// TwinCAT 3 PLC project PLC
// ProgramVersion: 3.1.4023.0
// libraries:
//   Tc2_Standard, * (Beckhoff Automation GmbH)
//   Tc2_System, * (Beckhoff Automation GmbH)
//   Tc3_Module, * (Beckhoff Automation GmbH)
// project tree:
//   / PlcTask.TcTTO
//   POUs/ MAIN.TcPOU
//   DUTs/IO/PdoEntries/ Status_B8381171.TcDUT, Status_182674C6.TcDUT, Status_7097155E.TcDUT, Control_DAEE1D52.TcDUT, Control_F189B737.TcDUT, Control_7786EF9F.TcDUT, Status_70E023F8.TcDUT, Control_A8DDCD82.TcDUT, Status_F2CE6D91.TcDUT, Status_B0753356.TcDUT, Status_68C33E99.TcDUT, Status_ACC8459F.TcDUT, Status_C03E2495.TcDUT, Status_D8D782C3.TcDUT, Control_6EF2C5D0.TcDUT, Status_3E6F3FF3.TcDUT, Status_3D84275F.TcDUT, Ctrl_1EFB4D3B.TcDUT, Status_B6795845.TcDUT, Control_C948E0F2.TcDUT, Status_8CBE219F.TcDUT, Status_1E008DB9.TcDUT, Control_5FD4673D.TcDUT, Status_3035BE2E.TcDUT, Status_2569232E.TcDUT, Control_FF5AB9B2.TcDUT, FSOE_1F44E1B4.TcDUT, FSOE_9A7ED3DD.TcDUT, FSOE_9F04885D.TcDUT, FSOE_87848461.TcDUT, FSOE_BBC930F7.TcDUT, FSOE_D1C9D1EA.TcDUT, FSOE_D94E700C.TcDUT, FSOE_1DB604F4.TcDUT, FSOE_046F804E.TcDUT, FSOE_2DC96D31.TcDUT
//   DUTs/IO/PDOs/ InfoData_6F19DB2B.TcDUT, WcState_0B2B16F9.TcDUT, InfoData_32EB74EA.TcDUT, Channel_830843C1.TcDUT, WcState_9091E0EB.TcDUT, Channel_42CA91F7.TcDUT, PWM_Outputs_Channel_4C6289CD.TcDUT, PTO_Status_E0EB10E8.TcDUT, ENC_Status_compact_3C6E2C44.TcDUT, PLS_Status_Channel_70E7A1E2.TcDUT, PTO_Control_9287F8E4.TcDUT, PTO_Target_compact_5C359F7D.TcDUT, ENC_Control_compact_2E82BC43.TcDUT, PLS_Control_compact_Channel_CD6E44DE.TcDUT, PTO_Status_Channel_E0EB10E8.TcDUT, ENC_Status_Channel_A9252C48.TcDUT, PTO_Control_Channel_9287F8E4.TcDUT, PTO_Target_Channel_1F6D5BC6.TcDUT, ENC_Control_Channel_686BB9DC.TcDUT, AI_Standard_Channel_4A394481.TcDUT, AI_Standard_Channel_A8DF64E3.TcDUT, RTD_Inputs_Channel_9575FEA1.TcDUT, TC_Channel_9575FEA1.TcDUT, AO_Output_Channel_BA7EBB7C.TcDUT, SSI_Inputs_Channel_0E3D8E33.TcDUT, SSI_Inputs_Channel_EDA16284.TcDUT, ENC_Status_compact_7D3464F3.TcDUT, ENC_Control_compact_21E2D14D.TcDUT, ENC_Inputs_B3536485.TcDUT, ENC_Inputs_24B63C53.TcDUT, ENC_Outputs_21E2D14D.TcDUT, COM_Inputs_Channel_3801C95E.TcDUT, COM_Outputs_Channel_EADA2E0D.TcDUT, DeviceState_Inputs_Device_A1210598.TcDUT, DeviceState_Inputs_4751FF76.TcDUT, InfoData_90184F0C.TcDUT, Module_1_DeviceState_Inputs_Device_5322301C.TcDUT, Module_2_DeviceState_Inputs_BD6C7035.TcDUT, STM_Status_36ED096F.TcDUT, STM_Control_5A8B5016.TcDUT, STM_Velocity_A47A3F41.TcDUT, InfoData_6538CF5F.TcDUT, ENC_Status_compact_4D066E1A.TcDUT, STM_Status_DE0D6B37.TcDUT, STM_Control_BA4CE352.TcDUT, ENC_Status_compact_Channel_DC559AB0.TcDUT, DCM_Status_Channel_36ED096F.TcDUT, ENC_Control_compact_Channel_2E82BC43.TcDUT, DCM_Control_Channel_5A8B5016.TcDUT, DCM_Velocity_Channel_A47A3F41.TcDUT, InfoData_939F71B6.TcDUT, FB_Position_3FA094ED.TcDUT, DRV_Statusword_9B36FDFC.TcDUT, DRV_Controlword_F3F14721.TcDUT, DRV_Target_velocity_08A9583B.TcDUT, InfoData_96C94FAE.TcDUT, InfoData_6185D47C.TcDUT, DS402_Statusword_9B36FDFC.TcDUT, DS402_Position_actual_value_07DC4C74.TcDUT, DS402_Controlword_F3F14721.TcDUT, DS402_Target_velocity_08A9583B.TcDUT, InfoData_8300A75E.TcDUT, DCM_Status_Channel_45521CDC.TcDUT, DCM_Outputs_Channel_F77F51CE.TcDUT, DRV_Following_error_actual_value_5AA320BF.TcDUT, DRV_Target_position_05240F14.TcDUT, Status_Uo_B8D9F2FA.TcDUT, BCT_Inputs_8E55234D.TcDUT, BCT_Inputs_4B987895.TcDUT, BCT_Inputs_8B1D510C.TcDUT, BCT_Inputs_7ACE8FA6.TcDUT, FSoE_Inputs_8952FEF0.TcDUT, FSoE_Outputs_7E672439.TcDUT, FIELDVOLTAGE_Field_Voltage_Status_9DC7C349.TcDUT, FSLOGIC_Inputs_EEE9388E.TcDUT, EMPTY_STRUCTURE.TcDUT, Module_1_FSOE_5515F18A.TcDUT, Module_2_DEVICEIO_5FA6B4E7.TcDUT, Module_3_FSLOGIC_DEAB4522.TcDUT, FSoE_Inputs_C661B78A.TcDUT, FSoE_Outputs_E138FCB5.TcDUT, Module_1_FSOE_18ED951F.TcDUT, FSoE_Inputs_8A5FBAF8.TcDUT, FSoE_Outputs_1F40D103.TcDUT, Outputs_7EDA7A42.TcDUT, WcState_B516A264.TcDUT, Module_1_FSOE_9FCACE14.TcDUT, Module_2_FSOUT_5A5AEBA4.TcDUT, Module_3_DEVICEIO_5FA6B4E7.TcDUT, Module_4_FSLOGIC_DEAB4522.TcDUT, FSoE_Inputs_15C2E7B1.TcDUT, FSoE_Outputs_C9D9BEFD.TcDUT, Module_1_FSOE_212A0B66.TcDUT, FSoE_Inputs_939ABF3D.TcDUT, FSoE_Outputs_2DD09AA7.TcDUT, Outputs_FB9F3520.TcDUT, Module_1_FSOE_7F12D292.TcDUT, Module_2_FSOUT_9813A38E.TcDUT, InfoData_E68C61CD.TcDUT, InfoData_2A97D6CF.TcDUT, Inputs_25A0042B.TcDUT, Outputs_2397A10E.TcDUT
//   DUTs/IO/Boxes/ EK1100_1FC0878B.TcDUT, EK1122_1FC0878B.TcDUT, EJ1100_1FC0878B.TcDUT, EJ1101_D4DF6A22.TcDUT, EJ1008_78E8D3DD.TcDUT, EJ1128_78E8D3DD.TcDUT, EJ1809_32157CFD.TcDUT, EJ1819_32157CFD.TcDUT, EJ1859_7699BCF6.TcDUT, EJ1889_32157CFD.TcDUT, EJ1122_1FC0878B.TcDUT, EJ2008_E2806B95.TcDUT, EJ2128_E2806B95.TcDUT, EJ2502_FE2154F7.TcDUT, EJ2521_E6A3E301.TcDUT, EJ2522_EF4C90EB.TcDUT, EJ2809_2B6483BD.TcDUT, EJ2889_2B6483BD.TcDUT, EJ3004_C4269E32.TcDUT, EJ3048_335F857B.TcDUT, EJ3058_335F857B.TcDUT, EJ3068_335F857B.TcDUT, EJ3104_DCC78662.TcDUT, EJ3108_335F857B.TcDUT, EJ3108_35AE5324.TcDUT, EJ3202_27F12237.TcDUT, EJ3214_8BBE23EA.TcDUT, EJ3255_1972F7C0.TcDUT, EJ3318_BD104D88.TcDUT, EJ4002_11E38659.TcDUT, EJ4002_5AE37D91.TcDUT, EJ4004_AB92710E.TcDUT, EJ4008_4E77D882.TcDUT, EJ4018_4E77D882.TcDUT, EJ4024_AB92710E.TcDUT, EJ4132_11E38659.TcDUT, EJ4134_15C7AA14.TcDUT, EJ5002_6DCBC4C0.TcDUT, EJ5002_31A396E2.TcDUT, EJ5101_7476E948.TcDUT, EJ5151_905C5FD8.TcDUT, EJ6002_D5B468BD.TcDUT, EJ6224_98EF2419.TcDUT, EJ7031_022B4804.TcDUT, EJ7037_3E4BEAEF.TcDUT, EJ7041_022B4804.TcDUT, EJ7047_3E4BEAEF.TcDUT, EJ7342_2AE9C6B3.TcDUT, EJ7211_CE650BCF.TcDUT, EJ7211_FC4732E8.TcDUT, EJ7211_7BF21317.TcDUT, EJ7211_B7F6AF53.TcDUT, EJ7334_80FE8C13.TcDUT, EJ7411_236AD61B.TcDUT, EJ9001_1FC0878B.TcDUT, EJ9505_19A4723D.TcDUT, EJ9576_6D7359CA.TcDUT, EJ9576_85AB5804.TcDUT, EJ9576_1017F4A5.TcDUT, EJ9576_C42142C6.TcDUT, EJ9400_B5091FDC.TcDUT, EJ9404_A60D6900.TcDUT, EJ1914_0821024F.TcDUT, EJ1918_57845E79.TcDUT, EJ1957_9A95FC59.TcDUT, EJ2914_475777A0.TcDUT, EJ2918_B661C90A.TcDUT, EJ6910_CD4DE200.TcDUT
//   DUTs/IO/Devices/ SyncUnitTask_2D604ED5.TcDUT, SyncUnitTasks_6FEB8257.TcDUT, SyncUnits_99E584AF.TcDUT
//   DUTs/IO/Topology/ Beckhoff_EJ1xxxEK1122_25307691.TcDUT, Beckhoff_EJ1xxx_8ABA4DFB.TcDUT, Beckhoff_EJ2xxxEK1122_536A6829.TcDUT, Beckhoff_EJ2xxx_F745D3BC.TcDUT, Beckhoff_EJ3xxxEK1122_1A5DA9A5.TcDUT, Beckhoff_EJ3xxx_05F253C1.TcDUT, Beckhoff_EJ4xxxEK1122_E11BF0B6.TcDUT, Beckhoff_EJ4xxx_77B5C5A6.TcDUT, Beckhoff_EJ5xxxEK1122_A82C313A.TcDUT, Beckhoff_EJ5xxx_E1A62FB7.TcDUT, Beckhoff_EJ6xxxEK1122_737473AE.TcDUT, Beckhoff_EJ6xxx_D380D5DE.TcDUT, Beckhoff_EJ7xxxEK1122_3A43B222.TcDUT, Beckhoff_EJ7xxx_D0F87F47.TcDUT, Beckhoff_EJ9xxxEK1122_C80E1DB3.TcDUT, Beckhoff_EJ9xxx_428E1E12.TcDUT, Beckhoff_EJx9xxEK1122_EEA9E9F5.TcDUT, Beckhoff_EJx9xx_66D9432D.TcDUT, EtherCAT_Master_EJxxxx_F8B494BA.TcDUT
//   DUTs/IO/Base/ EtcSlaveBase_82538BE2.TcDUT, EtcSlaveBase_82538BE2.TcDUT, EtcSlaveBase_82538BE2.TcDUT, EtcSlaveTerminalBase_947E5A46.TcDUT, EtcSlaveBoxBase_77A0E4A7.TcDUT, EtcSlaveEndTerminalBase_866C7F0C.TcDUT, InputBase_8311D824.TcDUT, OutputBase_10CEE7DE.TcDUT, EtcMasterBase_62654B43.TcDUT
//   GVLs/ GVL_iXlinker.TcGVL
// real-time tasks:
//   TASK PlcTask: cycle T#10ms, priority 20, ADS port 350
// I/O:
//   DEVICE EtherCAT_Master_EJxxxx, AmsNetId 172.20.30.238.7.1
//     Beckhoff EJ1xxx [EK1100 EtherCAT Coupler (2A E-Bus)]
//       Beckhoff EJ1xxxEK1122 [EK1122 2 port EtherCAT junction]
//         Beckhoff EJ1xxxsub EK1100 [EK1100 EtherCAT Coupler (2A E-Bus)]
//         A_0001(EJ1100-0000-0018) [EJ1100 EtherCAT Coupler (2.2A E-Bus)]
//         A_0002(EJ1101-0022-0016) [EJ1101-0022 EtherCAT Coupler (ID switch)]
//       A_0004(EJ1008-0000-0017) [EJ1008 8Ch. Dig. Input 24V, 3ms]
//       A_0005(EJ1128-0000-0016) [EJ1128 8Ch. Dig. Input 5V / 3.3V DC, 0.05µs]
//       A_0006(EJ1809-0000-0017) [EJ1809 16Ch. Dig. Input 24V, 3ms]
//       A_0007(EJ1819-0000-0017) [EJ1819 16Ch. Dig. Input 24V, 10µs]
//       A_0008(EJ1859-0000-0017) [EJ1859 8Ch. Dig. Input 24V, 3ms, 8Ch. Dig. Output 24V, 0.5A]
//       A_0009(EJ1889-0000-0017) [EJ1889 16Ch. Dig. Input 24V, 3ms, negative]
//       A_0003(EJ1122-0000-0016) [EJ1122 2 port EtherCAT junction]
//     Beckhoff EJ2xxx [EK1100 EtherCAT Coupler (2A E-Bus)]
//       Beckhoff EJ2xxxEK1122 [EK1122 2 port EtherCAT junction]
//         Beckhoff EJ2xxxsub EK1100 [EK1100 EtherCAT Coupler (2A E-Bus)]
//       A_0001(EJ2008-0000-0017) [EJ2008 8Ch. Dig. Output 24V, 0.5A]
//       A_0002(EJ2008-0000-0018) [EJ2008 8Ch. Dig. Output 24V, 0.5A]
//       A_0003(EJ2128-0000-0016) [EJ2128 8Ch. Dig. Output 5V/3.3V, 20mA]
//       A_0004(EJ2502-0000-0023) [EJ2502 2Ch. PWM output, 24V]
//       A_0005(EJ2502-0000-0024) [EJ2502 2Ch. PWM output, 24V]
//       A_0006(EJ2521-0224-0016) [EJ2521-0224 1Ch. Pulse Train 24V DC Output Capture/Compare]
//       A_0007(EJ2522-0000-0022) [EJ2522 2Ch. Pulse Train Output]
//       A_0008(EJ2809-0000-0017) [EJ2809 16Ch. Dig. Output 24V, 0.5A]
//       A_0009(EJ2889-0000-0016) [EJ2889 16Ch. Dig. Output 24V, 0.5A, negative]
//       A_0010(EJ2889-0000-0017) [EJ2889 16Ch. Dig. Output 24V, 0.5A, negative]
//     Beckhoff EJ3xxx [EK1100 EtherCAT Coupler (2A E-Bus)]
//       Beckhoff EJ3xxxEK1122 [EK1122 2 port EtherCAT junction]
//         Beckhoff EJ3xxxsub EK1100 [EK1100 EtherCAT Coupler (2A E-Bus)]
//       A_0001(EJ3004-0000-0019) [EJ3004 4Ch. Ana. Input +/-10V]
//       A_0002(EJ3004-0000-0020) [EJ3004 4Ch. Ana. Input +/-10V]
//       A_0003(EJ3004-0000-0021) [EJ3004 4Ch. Ana. Input +/-10V]
//       A_0004(EJ3048-0000-0020) [EJ3048 8Ch. Ana. Input 0-20mA]
//       A_0005(EJ3058-0000-0020) [EJ3058 8Ch. Ana. Input 4-20mA]
//       A_0006(EJ3068-0000-0020) [EJ3068 8Ch. Ana. Input 0-10V]
//       A_0007(EJ3068-0000-0021) [EJ3068 8Ch. Ana. Input 0-10V]
//       A_0008(EJ3104-0000-0019) [EJ3104 4Ch. Ana. Input +/-10V DIFF]
//       A_0009(EJ3104-0000-0020) [EJ3104 4Ch. Ana. Input +/-10V DIFF]
//       A_0010(EJ3104-0000-0021) [EJ3104 4Ch. Ana. Input +/-10V DIFF]
//       A_0011(EJ3108-0000-0017) [EJ3108 8Ch. Ana. Input +/-10V]
//       A_0012(EJ3108-0000-0018) [EJ3108 8Ch. Ana. Input +/-10V]
//       A_0013(EJ3108-0000-0019) [EJ3108 8Ch. Ana. Input +/-10V]
//       A_0014(EJ3202-0000-0019) [EJ3202 2Ch. Ana. Input PT100 (RTD)]
//       A_0015(EJ3202-0000-0020) [EJ3202 2Ch. Ana. Input PT100 (RTD)]
//       A_0016(EJ3202-0000-0021) [EJ3202 2Ch. Ana. Input PT100 (RTD)]
//       A_0017(EJ3214-0000-0016) [EJ3214 4Ch. Ana. Input PT100 (RTD)]
//       A_0018(EJ3255-0000-0023) [EJ3255 5Ch. potentiometer measurement with sensor supply]
//       A_0019(EJ3318-0000-0017) [EJ3318 8Ch. Ana Input Thermocouple (TC)]
//     Beckhoff EJ4xxx [EK1100 EtherCAT Coupler (2A E-Bus)]
//       Beckhoff EJ4xxxEK1122 [EK1122 2 port EtherCAT junction]
//         Beckhoff EJ4xxxsub EK1100 [EK1100 EtherCAT Coupler (2A E-Bus)]
//       A_0001(EJ4002-0000-0017) [EJ4002 2Ch. Ana. Output 0-10V, 12bit]
//       A_0002(EJ4002-0000-0018) [EJ4002 2Ch. Ana. Output 0-10V, 12bit]
//       A_0003(EJ4004-0000-0020) [EJ4004 4Ch. Ana. Output 0-10V, 12bit]
//       A_0004(EJ4008-0000-0020) [EJ4008 8Ch. Ana. Output 0-10V, 12bit]
//       A_0005(EJ4018-0000-0016) [EJ4018 8Ch. Ana. Output 0-20mA, 12bit]
//       A_0006(EJ4024-0000-0020) [EJ4024 4Ch. Ana. Output 4-20mA, 12bit]
//       A_0007(EJ4132-0000-0019) [EJ4132 2Ch. Ana. Output -10/+10V, 16bit]
//       A_0008(EJ4134-0000-0019) [EJ4134 4Ch. Ana. Output -10/+10V, 16bit]
//       A_0009(EJ4134-0000-0020) [EJ4134 4Ch. Ana. Output -10/+10V, 16bit]
//     Beckhoff EJ5xxx [EK1100 EtherCAT Coupler (2A E-Bus)]
//       Beckhoff EJ5xxxEK1122 [EK1122 2 port EtherCAT junction]
//         Beckhoff EJ5xxxsub EK1100 [EK1100 EtherCAT Coupler (2A E-Bus)]
//       A_0001(EJ5002-0000-0016) [EJ5002 2Ch. SSI Encoder]
//       A_0002(EJ5002-0000-0017) [EJ5002 2Ch. SSI Encoder]
//       A_0003(EJ5101-0000-0016) [EJ5101 1Ch. Inc. Encoder 5V]
//       A_0004(EJ5151-0000-0016) [EJ5151 1Ch. Inc. Encoder]
//     Beckhoff EJ6xxx [EK1100 EtherCAT Coupler (2A E-Bus)]
//       Beckhoff EJ6xxxEK1122 [EK1122 2 port EtherCAT junction]
//         Beckhoff EJ6xxxsub EK1100 [EK1100 EtherCAT Coupler (2A E-Bus)]
//       A_0001(EJ6002-0000-0016) [EJ6002 Interface 2Ch. (RS232/RS485/RS422)]
//       A_0002(EJ6224-0000-0016) [EJ6224 (IO Link Master)]
//         modules: Module 1 (DeviceState Inputs Device), Module 2 (DeviceState Inputs), Module 3 (empty), Module 4 (empty), Module 5 (empty), Module 6 (empty)
//       A_0003(EJ6224-0090-0016) [EJ6224-0090 (IO Link Master, TwinSAFE SC)]
//         modules: Module 1 (DeviceState Inputs Device), Module 2 (DeviceState Inputs), Module 3 (empty), Module 4 (empty), Module 5 (empty), Module 6 (empty)
//     Beckhoff EJ7xxx [EK1100 EtherCAT Coupler (2A E-Bus)]
//       Beckhoff EJ7xxxEK1122 [EK1122 2 port EtherCAT junction]
//         Beckhoff EJ7xxxsub EK1100 [EK1100 EtherCAT Coupler (2A E-Bus)]
//       A_0001(EJ7031-0000-0026) [EJ7031 1Ch. Stepper motor output stage (24V, 1.5A)]
//       A_0002(EJ7037-0000-0020) [EJ7037 1Ch. Stepper motor output stage (24V, 1.5A)]
//       A_0003(EJ7041-0052-0016) [EJ7041-0052 1Ch. Stepper motor output stage (50V, 5A)]
//       A_0004(EJ7047-0000-0018) [EJ7047 1Ch. Stepper motor output stage (50V, 5A)]
//       A_0005(EJ7047-0000-0019) [EJ7047 1Ch. Stepper motor output stage (50V, 5A)]
//       A_0006(EJ7047-0000-0020) [EJ7047 1Ch. Stepper motor output stage (50V, 5A)]
//       A_0007(EJ7342-0000-0019) [EJ7342 2Ch. DC motor output stage (50V, 3.5A)]
//       A_0008(EJ7342-0000-0020) [EJ7342 2Ch. DC motor output stage (50V, 3.5A)]
//       A_0009(EJ7211-0010-0026) [EJ7211-0010 1Ch. MDP742 Servo motor output stage with OCT (50V, 4.5A RMS)]
//       A_0010(EJ7211-0010-0027) [EJ7211-0010 1Ch. MDP742 Servo motor output stage with OCT (50V, 4.5A RMS)]
//       A_0011(EJ7211-0010-0028) [EJ7211-0010 1Ch. MDP742 Servo motor output stage with OCT (50V, 4.5A RMS)]
//       A_0012(EJ7211-0010-0029) [EJ7211-0010 1Ch. MDP742 Servo motor output stage with OCT (50V, 4.5A RMS)]
//       A_0013(EJ7211-0010-0030) [EJ7211-0010 1Ch. MDP742 Servo motor output stage with OCT (50V, 4.5A RMS)]
//       A_0014(EJ7211-0010-0031) [EJ7211-0010 1Ch. MDP742 Servo motor output stage with OCT (50V, 4.5A RMS)]
//       A_0015(EJ7211-0010-0032) [EJ7211-0010 1Ch. MDP742 Servo motor output stage with OCT (50V, 4.5A RMS)]
//       A_0016(EJ7211-0011-0026) [EJ7211-0011 1Ch. DS402 Servo motor output stage with OCT (50V, 4.5A RMS)]
//       A_0017(EJ7211-0011-0027) [EJ7211-0011 1Ch. DS402 Servo motor output stage with OCT (50V, 4.5A RMS)]
//       A_0018(EJ7211-0011-0028) [EJ7211-0011 1Ch. DS402 Servo motor output stage with OCT (50V, 4.5A RMS)]
//       A_0019(EJ7211-0011-0029) [EJ7211-0011 1Ch. DS402 Servo motor output stage with OCT (50V, 4.5A RMS)]
//       A_0020(EJ7211-0011-0030) [EJ7211-0011 1Ch. DS402 Servo motor output stage with OCT (50V, 4.5A RMS)]
//       A_0021(EJ7211-0011-0031) [EJ7211-0011 1Ch. DS402 Servo motor output stage with OCT (50V, 4.5A RMS)]
//       A_0022(EJ7211-0011-0032) [EJ7211-0011 1Ch. DS402 Servo motor output stage with OCT (50V, 4.5A RMS)]
//       A_0023(EJ7211-9414-0029) [EJ7211-9414 1Ch. MDP742 Servo motor output stage with OCT (50V, 4.5A RMS) , TwinSAFE SC]
//       A_0024(EJ7211-9414-0030) [EJ7211-9414 1Ch. MDP742 Servo motor output stage with OCT (50V, 4.5A RMS) , TwinSAFE SC]
//       A_0025(EJ7211-9414-0031) [EJ7211-9414 1Ch. MDP742 Servo motor output stage with OCT (50V, 4.5A RMS) , TwinSAFE SC]
//       A_0026(EJ7211-9414-0032) [EJ7211-9414 1Ch. MDP742 Servo motor output stage with OCT (50V, 4.5A RMS) , TwinSAFE SC]
//       A_0027(EJ7211-9415-0029) [EJ7211-9415 1Ch. DS402 Servo motor output stage with OCT (50V, 4.5A RMS), TwinSAFE SC]
//       A_0028(EJ7211-9415-0030) [EJ7211-9415 1Ch. DS402 Servo motor output stage with OCT (50V, 4.5A RMS), TwinSAFE SC]
//       A_0029(EJ7211-9415-0031) [EJ7211-9415 1Ch. DS402 Servo motor output stage with OCT (50V, 4.5A RMS), TwinSAFE SC]
//       A_0030(EJ7211-9415-0032) [EJ7211-9415 1Ch. DS402 Servo motor output stage with OCT (50V, 4.5A RMS), TwinSAFE SC]
//       A_0031(EJ7334-0008-0016) [EJ7334-0008 4 Ch. Bi-/8 Ch. Unidirectional DC motor output stage (24 V, 8 A overall current)]
//       A_0032(EJ7411-0000-0018) [EJ7411 BLDC Terminal with incremental encoder/Hall, 50 V DC, 4.5 A]
//     Beckhoff EJ9xxx [EK1100 EtherCAT Coupler (2A E-Bus)]
//       Beckhoff EJ9xxxEK1122 [EK1122 2 port EtherCAT junction]
//         Beckhoff EJ9xxxsub EK1100 [EK1100 EtherCAT Coupler (2A E-Bus)]
//       A_0001(EJ9001-0000-0016) [EJ9001 placeholder module]
//       A_0002(EJ9505-0000-0016) [EJ9505 Power supply module 5V]
//       A_0003(EJ9576-0000-0018) [EJ9576 Brake chopper terminal]
//       A_0004(EJ9576-0000-0019) [EJ9576 Brake chopper terminal]
//       A_0005(EJ9576-0000-0020) [EJ9576 Brake chopper terminal]
//       A_0006(EJ9576-0000-0022) [EJ9576 Brake chopper terminal]
//       A_0007 (EJ9400-0000) [EJ9400-0000 Power supply module 2,5A]
//       A_0008 (EJ9404-0000) [EJ9404-0000 Power supply module 12A]
//     Beckhoff EJx9xx [EK1100 EtherCAT Coupler (2A E-Bus)]
//       Beckhoff EJx9xxEK1122 [EK1122 2 port EtherCAT junction]
//         Beckhoff EJx9xxsub EK1100 [EK1100 EtherCAT Coupler (2A E-Bus)]
//       A_0001(EJ1914-0000-0017) [EJ1914-0000-0017]
//         modules: Module 1 (FSOE), Module 2 (DEVICEIO), Module 3 (FSLOGIC)
//       A_0002(EJ1914-0000-0018) [EJ1914, 4Ch. Safety Input 24V, TwinSAFE]
//         modules: Module 1 (FSOE), Module 2 (DEVICEIO), Module 3 (FSLOGIC)
//       A_0003(EJ1918-0000-0017) [EJ1918-0000-0017]
//         modules: Module 1 (FSOE), Module 2 (DEVICEIO), Module 3 (FSLOGIC)
//       A_0004(EJ1918-0000-0018) [EJ1918, 8Ch. Safety Input 24V, TwinSAFE]
//         modules: Module 1 (FSOE), Module 2 (DEVICEIO), Module 3 (FSLOGIC)
//       A_0005(EJ1957-0000-0017) [EJ1957-0000-0017]
//         modules: Module 1 (FSOE), Module 2 (FSOUT), Module 3 (DEVICEIO), Module 4 (FSLOGIC)
//       A_0006(EJ1957-0000-0018) [EJ1957, 8Ch. Safety Input 24V, 4Ch. Safety Output 24V, 0.5A, TwinSAFE]
//         modules: Module 1 (FSOE), Module 2 (FSOUT), Module 3 (DEVICEIO), Module 4 (FSLOGIC)
//       A_0007(EJ2914-0000-0017) [EJ2914-0000-0017]
//         modules: Module 1 (FSOE), Module 2 (FSOUT), Module 3 (DEVICEIO), Module 4 (FSLOGIC)
//       A_0008(EJ2914-0000-0018) [EJ2914, 4Ch. Safety Output 24V, 0.5A, TwinSAFE]
//         modules: Module 1 (FSOE), Module 2 (FSOUT), Module 3 (DEVICEIO), Module 4 (FSLOGIC)
//       A_0009(EJ2918-0000-0017) [EJ2918-0000-0017]
//         modules: Module 1 (FSOE), Module 2 (FSOUT), Module 3 (DEVICEIO), Module 4 (FSLOGIC)
//       A_0010(EJ2918-0000-0018) [EJ2918, 8Ch. Safety Output 24V, 0.5A, TwinSAFE]
//         modules: Module 1 (FSOE), Module 2 (FSOUT), Module 3 (DEVICEIO), Module 4 (FSLOGIC)
//       A_0011(EJ6910-0000-0018) [EJ6910, TwinSAFE PLC]
//       A_0012(EJ6910-0000-0020) [EJ6910, TwinSAFE PLC]
// variable links:
//   PLC/PLC Instance <-> EtherCAT Master EJxxxx/Beckhoff EJ1xxx
//     PlcTask Inputs/GVL_iXlinker.EtherCAT_Master_EJxxxx.Beckhoff_EJ1xxx.InfoData.State <-> InfoData/State
//   PLC/PLC Instance <-> EtherCAT Master EJxxxx/Beckhoff EJ1xxx/Beckhoff EJ1xxxEK1122
//     PlcTask Inputs/GVL_iXlinker.EtherCAT_Master_EJxxxx.Beckhoff_EJ1xxx.Beckhoff_EJ1xxxEK1122.InfoData.State <-> InfoData/State
//   PLC/PLC Instance <-> EtherCAT Master EJxxxx/Beckhoff EJ1xxx/Beckhoff EJ1xxxEK1122/Beckhoff EJ1xxxsub EK1100
//     PlcTask Inputs/GVL_iXlinker.EtherCAT_Master_EJxxxx.Beckhoff_EJ1xxx.Beckhoff_EJ1xxxEK1122.Beckhoff_EJ1xxxsub_EK1100.InfoData.State <-> InfoData/State
//   PLC/PLC Instance <-> EtherCAT Master EJxxxx/Beckhoff EJ1xxx/Beckhoff EJ1xxxEK1122/A_0001(EJ1100-0000-0018)
//     PlcTask Inputs/GVL_iXlinker.EtherCAT_Master_EJxxxx.Beckhoff_EJ1xxx.Beckhoff_EJ1xxxEK1122.A_0001_EJ1100_0000_0018.InfoData.State <-> InfoData/State
//   PLC/PLC Instance <-> EtherCAT Master EJxxxx/Beckhoff EJ1xxx/Beckhoff EJ1xxxEK1122/A_0002(EJ1101-0022-0016)
//     PlcTask Inputs/GVL_iXlinker.EtherCAT_Master_EJxxxx.Beckhoff_EJ1xxx.Beckhoff_EJ1xxxEK1122.A_0002_EJ1101_0022_0016.WcState.WcState <-> WcState/WcState
//     PlcTask Inputs/GVL_iXlinker.EtherCAT_Master_EJxxxx.Beckhoff_EJ1xxx.Beckhoff_EJ1xxxEK1122.A_0002_EJ1101_0022_0016.InfoData.AdsAddr <-> InfoData/AdsAddr
//     PlcTask Inputs/GVL_iXlinker.EtherCAT_Master_EJxxxx.Beckhoff_EJ1xxx.Beckhoff_EJ1xxxEK1122.A_0002_EJ1101_0022_0016.InfoData.State <-> InfoData/State
//   PLC/PLC Instance <-> EtherCAT Master EJxxxx/Beckhoff EJ1xxx/A_0004(EJ1008-0000-0017)
//     PlcTask Inputs/GVL_iXlinker.EtherCAT_Master_EJxxxx.Beckhoff_EJ1xxx.A_0004_EJ1008_0000_0017.Channel_1.Input <-> Channel 1/Input
//     PlcTask Inputs/GVL_iXlinker.EtherCAT_Master_EJxxxx.Beckhoff_EJ1xxx.A_0004_EJ1008_0000_0017.Channel_2.Input <-> Channel 2/Input
//     PlcTask Inputs/GVL_iXlinker.EtherCAT_Master_EJxxxx.Beckhoff_EJ1xxx.A_0004_EJ1008_0000_0017.Channel_3.Input <-> Channel 3/Input
//     PlcTask Inputs/GVL_iXlinker.EtherCAT_Master_EJxxxx.Beckhoff_EJ1xxx.A_0004_EJ1008_0000_0017.Channel_4.Input <-> Channel 4/Input
//     PlcTask Inputs/GVL_iXlinker.EtherCAT_Master_EJxxxx.Beckhoff_EJ1xxx.A_0004_EJ1008_0000_0017.Channel_5.Input <-> Channel 5/Input
//     PlcTask Inputs/GVL_iXlinker.EtherCAT_Master_EJxxxx.Beckhoff_EJ1xxx.A_0004_EJ1008_0000_0017.Channel_6.Input <-> Channel 6/Input
//     PlcTask Inputs/GVL_iXlinker.EtherCAT_Master_EJxxxx.Beckhoff_EJ1xxx.A_0004_EJ1008_0000_0017.Channel_7.Input <-> Channel 7/Input
//     PlcTask Inputs/GVL_iXlinker.EtherCAT_Master_EJxxxx.Beckhoff_EJ1xxx.A_0004_EJ1008_0000_0017.Channel_8.Input <-> Channel 8/Input
//     PlcTask Inputs/GVL_iXlinker.EtherCAT_Master_EJxxxx.Beckhoff_EJ1xxx.A_0004_EJ1008_0000_0017.WcState.WcState <-> WcState/WcState
//     PlcTask Inputs/GVL_iXlinker.EtherCAT_Master_EJxxxx.Beckhoff_EJ1xxx.A_0004_EJ1008_0000_0017.WcState.InputToggle <-> WcState/InputToggle
//     PlcTask Inputs/GVL_iXlinker.EtherCAT_Master_EJxxxx.Beckhoff_EJ1xxx.A_0004_EJ1008_0000_0017.InfoData.State <-> InfoData/State
//   PLC/PLC Instance <-> EtherCAT Master EJxxxx/Beckhoff EJ1xxx/A_0005(EJ1128-0000-0016)
//     PlcTask Inputs/GVL_iXlinker.EtherCAT_Master_EJxxxx.Beckhoff_EJ1xxx.A_0005_EJ1128_0000_0016.Channel_1.Input <-> Channel 1/Input
//     PlcTask Inputs/GVL_iXlinker.EtherCAT_Master_EJxxxx.Beckhoff_EJ1xxx.A_0005_EJ1128_0000_0016.Channel_2.Input <-> Channel 2/Input
//     PlcTask Inputs/GVL_iXlinker.EtherCAT_Master_EJxxxx.Beckhoff_EJ1xxx.A_0005_EJ1128_0000_0016.Channel_3.Input <-> Channel 3/Input
//     PlcTask Inputs/GVL_iXlinker.EtherCAT_Master_EJxxxx.Beckhoff_EJ1xxx.A_0005_EJ1128_0000_0016.Channel_4.Input <-> Channel 4/Input
//     PlcTask Inputs/GVL_iXlinker.EtherCAT_Master_EJxxxx.Beckhoff_EJ1xxx.A_0005_EJ1128_0000_0016.Channel_5.Input <-> Channel 5/Input
//     PlcTask Inputs/GVL_iXlinker.EtherCAT_Master_EJxxxx.Beckhoff_EJ1xxx.A_0005_EJ1128_0000_0016.Channel_6.Input <-> Channel 6/Input
//     PlcTask Inputs/GVL_iXlinker.EtherCAT_Master_EJxxxx.Beckhoff_EJ1xxx.A_0005_EJ1128_0000_0016.Channel_7.Input <-> Channel 7/Input
//     PlcTask Inputs/GVL_iXlinker.EtherCAT_Master_EJxxxx.Beckhoff_EJ1xxx.A_0005_EJ1128_0000_0016.Channel_8.Input <-> Channel 8/Input
//     PlcTask Inputs/GVL_iXlinker.EtherCAT_Master_EJxxxx.Beckhoff_EJ1xxx.A_0005_EJ1128_0000_0016.WcState.WcState <-> WcState/WcState
//     PlcTask Inputs/GVL_iXlinker.EtherCAT_Master_EJxxxx.Beckhoff_EJ1xxx.A_0005_EJ1128_0000_0016.WcState.InputToggle <-> WcState/InputToggle
//     PlcTask Inputs/GVL_iXlinker.EtherCAT_Master_EJxxxx.Beckhoff_EJ1xxx.A_0005_EJ1128_0000_0016.InfoData.State <-> InfoData/State
//   PLC/PLC Instance <-> EtherCAT Master EJxxxx/Beckhoff EJ1xxx/A_0006(EJ1809-0000-0017)
//     PlcTask Inputs/GVL_iXlinker.EtherCAT_Master_EJxxxx.Beckhoff_EJ1xxx.A_0006_EJ1809_0000_0017.Channel_1.Input <-> Channel 1/Input
//     PlcTask Inputs/GVL_iXlinker.EtherCAT_Master_EJxxxx.Beckhoff_EJ1xxx.A_0006_EJ1809_0000_0017.Channel_2.Input <-> Channel 2/Input
//     PlcTask Inputs/GVL_iXlinker.EtherCAT_Master_EJxxxx.Beckhoff_EJ1xxx.A_0006_EJ1809_0000_0017.Channel_3.Input <-> Channel 3/Input
//     PlcTask Inputs/GVL_iXlinker.EtherCAT_Master_EJxxxx.Beckhoff_EJ1xxx.A_0006_EJ1809_0000_0017.Channel_4.Input <-> Channel 4/Input
//     PlcTask Inputs/GVL_iXlinker.EtherCAT_Master_EJxxxx.Beckhoff_EJ1xxx.A_0006_EJ1809_0000_0017.Channel_5.Input <-> Channel 5/Input
//     PlcTask Inputs/GVL_iXlinker.EtherCAT_Master_EJxxxx.Beckhoff_EJ1xxx.A_0006_EJ1809_0000_0017.Channel_6.Input <-> Channel 6/Input
//     PlcTask Inputs/GVL_iXlinker.EtherCAT_Master_EJxxxx.Beckhoff_EJ1xxx.A_0006_EJ1809_0000_0017.Channel_7.Input <-> Channel 7/Input
//     PlcTask Inputs/GVL_iXlinker.EtherCAT_Master_EJxxxx.Beckhoff_EJ1xxx.A_0006_EJ1809_0000_0017.Channel_8.Input <-> Channel 8/Input
//     PlcTask Inputs/GVL_iXlinker.EtherCAT_Master_EJxxxx.Beckhoff_EJ1xxx.A_0006_EJ1809_0000_0017.Channel_9.Input <-> Channel 9/Input
//     PlcTask Inputs/GVL_iXlinker.EtherCAT_Master_EJxxxx.Beckhoff_EJ1xxx.A_0006_EJ1809_0000_0017.Channel_10.Input <-> Channel 10/Input
//     PlcTask Inputs/GVL_iXlinker.EtherCAT_Master_EJxxxx.Beckhoff_EJ1xxx.A_0006_EJ1809_0000_0017.Channel_11.Input <-> Channel 11/Input
//     PlcTask Inputs/GVL_iXlinker.EtherCAT_Master_EJxxxx.Beckhoff_EJ1xxx.A_0006_EJ1809_0000_0017.Channel_12.Input <-> Channel 12/Input
//     PlcTask Inputs/GVL_iXlinker.EtherCAT_Master_EJxxxx.Beckhoff_EJ1xxx.A_0006_EJ1809_0000_0017.Channel_13.Input <-> Channel 13/Input
//     PlcTask Inputs/GVL_iXlinker.EtherCAT_Master_EJxxxx.Beckhoff_EJ1xxx.A_0006_EJ1809_0000_0017.Channel_14.Input <-> Channel 14/Input
//     PlcTask Inputs/GVL_iXlinker.EtherCAT_Master_EJxxxx.Beckhoff_EJ1xxx.A_0006_EJ1809_0000_0017.Channel_15.Input <-> Channel 15/Input
//     PlcTask Inputs/GVL_iXlinker.EtherCAT_Master_EJxxxx.Beckhoff_EJ1xxx.A_0006_EJ1809_0000_0017.Channel_16.Input <-> Channel 16/Input
//     PlcTask Inputs/GVL_iXlinker.EtherCAT_Master_EJxxxx.Beckhoff_EJ1xxx.A_0006_EJ1809_0000_0017.WcState.WcState <-> WcState/WcState
//     PlcTask Inputs/GVL_iXlinker.EtherCAT_Master_EJxxxx.Beckhoff_EJ1xxx.A_0006_EJ1809_0000_0017.WcState.InputToggle <-> WcState/InputToggle
//     PlcTask Inputs/GVL_iXlinker.EtherCAT_Master_EJxxxx.Beckhoff_EJ1xxx.A_0006_EJ1809_0000_0017.InfoData.State <-> InfoData/State
//   PLC/PLC Instance <-> EtherCAT Master EJxxxx/Beckhoff EJ1xxx/A_0007(EJ1819-0000-0017)
//     PlcTask Inputs/GVL_iXlinker.EtherCAT_Master_EJxxxx.Beckhoff_EJ1xxx.A_0007_EJ1819_0000_0017.Channel_1.Input <-> Channel 1/Input
//     PlcTask Inputs/GVL_iXlinker.EtherCAT_Master_EJxxxx.Beckhoff_EJ1xxx.A_0007_EJ1819_0000_0017.Channel_2.Input <-> Channel 2/Input
//     PlcTask Inputs/GVL_iXlinker.EtherCAT_Master_EJxxxx.Beckhoff_EJ1xxx.A_0007_EJ1819_0000_0017.Channel_3.Input <-> Channel 3/Input
//     PlcTask Inputs/GVL_iXlinker.EtherCAT_Master_EJxxxx.Beckhoff_EJ1xxx.A_0007_EJ1819_0000_0017.Channel_4.Input <-> Channel 4/Input
//     PlcTask Inputs/GVL_iXlinker.EtherCAT_Master_EJxxxx.Beckhoff_EJ1xxx.A_0007_EJ1819_0000_0017.Channel_5.Input <-> Channel 5/Input
//     PlcTask Inputs/GVL_iXlinker.EtherCAT_Master_EJxxxx.Beckhoff_EJ1xxx.A_0007_EJ1819_0000_0017.Channel_6.Input <-> Channel 6/Input
//     PlcTask Inputs/GVL_iXlinker.EtherCAT_Master_EJxxxx.Beckhoff_EJ1xxx.A_0007_EJ1819_0000_0017.Channel_7.Input <-> Channel 7/Input
//     PlcTask Inputs/GVL_iXlinker.EtherCAT_Master_EJxxxx.Beckhoff_EJ1xxx.A_0007_EJ1819_0000_0017.Channel_8.Input <-> Channel 8/Input
//     PlcTask Inputs/GVL_iXlinker.EtherCAT_Master_EJxxxx.Beckhoff_EJ1xxx.A_0007_EJ1819_0000_0017.Channel_9.Input <-> Channel 9/Input
//     PlcTask Inputs/GVL_iXlinker.EtherCAT_Master_EJxxxx.Beckhoff_EJ1xxx.A_0007_EJ1819_0000_0017.Channel_10.Input <-> Channel 10/Input
//     PlcTask Inputs/GVL_iXlinker.EtherCAT_Master_EJxxxx.Beckhoff_EJ1xxx.A_0007_EJ1819_0000_0017.Channel_11.Input <-> Channel 11/Input
//     PlcTask Inputs/GVL_iXlinker.EtherCAT_Master_EJxxxx.Beckhoff_EJ1xxx.A_0007_EJ1819_0000_0017.Channel_12.Input <-> Channel 12/Input
//     PlcTask Inputs/GVL_iXlinker.EtherCAT_Master_EJxxxx.Beckhoff_EJ1xxx.A_0007_EJ1819_0000_0017.Channel_13.Input <-> Channel 13/Input
//     PlcTask Inputs/GVL_iXlinker.EtherCAT_Master_EJxxxx.Beckhoff_EJ1xxx.A_0007_EJ1819_0000_0017.Channel_14.Input <-> Channel 14/Input
//     PlcTask Inputs/GVL_iXlinker.EtherCAT_Master_EJxxxx.Beckhoff_EJ1xxx.A_0007_EJ1819_0000_0017.Channel_15.Input <-> Channel 15/Input
//     PlcTask Inputs/GVL_iXlinker.EtherCAT_Master_EJxxxx.Beckhoff_EJ1xxx.A_0007_EJ1819_0000_0017.Channel_16.Input <-> Channel 16/Input
//     PlcTask Inputs/GVL_iXlinker.EtherCAT_Master_EJxxxx.Beckhoff_EJ1xxx.A_0007_EJ1819_0000_0017.WcState.WcState <-> WcState/WcState
//     PlcTask Inputs/GVL_iXlinker.EtherCAT_Master_EJxxxx.Beckhoff_EJ1xxx.A_0007_EJ1819_0000_0017.WcState.InputToggle <-> WcState/InputToggle
//     PlcTask Inputs/GVL_iXlinker.EtherCAT_Master_EJxxxx.Beckhoff_EJ1xxx.A_0007_EJ1819_0000_0017.InfoData.State <-> InfoData/State
//   PLC/PLC Instance <-> EtherCAT Master EJxxxx/Beckhoff EJ1xxx/A_0008(EJ1859-0000-0017)
//     PlcTask Inputs/GVL_iXlinker.EtherCAT_Master_EJxxxx.Beckhoff_EJ1xxx.A_0008_EJ1859_0000_0017.Channel_1.Input <-> Channel 1/Input
//     PlcTask Inputs/GVL_iXlinker.EtherCAT_Master_EJxxxx.Beckhoff_EJ1xxx.A_0008_EJ1859_0000_0017.Channel_2.Input <-> Channel 2/Input
//     PlcTask Inputs/GVL_iXlinker.EtherCAT_Master_EJxxxx.Beckhoff_EJ1xxx.A_0008_EJ1859_0000_0017.Channel_3.Input <-> Channel 3/Input
//     PlcTask Inputs/GVL_iXlinker.EtherCAT_Master_EJxxxx.Beckhoff_EJ1xxx.A_0008_EJ1859_0000_0017.Channel_4.Input <-> Channel 4/Input
//     PlcTask Inputs/GVL_iXlinker.EtherCAT_Master_EJxxxx.Beckhoff_EJ1xxx.A_0008_EJ1859_0000_0017.Channel_5.Input <-> Channel 5/Input
//     PlcTask Inputs/GVL_iXlinker.EtherCAT_Master_EJxxxx.Beckhoff_EJ1xxx.A_0008_EJ1859_0000_0017.Channel_6.Input <-> Channel 6/Input
//     PlcTask Inputs/GVL_iXlinker.EtherCAT_Master_EJxxxx.Beckhoff_EJ1xxx.A_0008_EJ1859_0000_0017.Channel_7.Input <-> Channel 7/Input
//     PlcTask Inputs/GVL_iXlinker.EtherCAT_Master_EJxxxx.Beckhoff_EJ1xxx.A_0008_EJ1859_0000_0017.Channel_8.Input <-> Channel 8/Input
//     PlcTask Outputs/GVL_iXlinker.EtherCAT_Master_EJxxxx.Beckhoff_EJ1xxx.A_0008_EJ1859_0000_0017.Channel_9.Output <-> Channel 9/Output
//     PlcTask Outputs/GVL_iXlinker.EtherCAT_Master_EJxxxx.Beckhoff_EJ1xxx.A_0008_EJ1859_0000_0017.Channel_10.Output <-> Channel 10/Output
//     PlcTask Outputs/GVL_iXlinker.EtherCAT_Master_EJxxxx.Beckhoff_EJ1xxx.A_0008_EJ1859_0000_0017.Channel_11.Output <-> Channel 11/Output
//     PlcTask Outputs/GVL_iXlinker.EtherCAT_Master_EJxxxx.Beckhoff_EJ1xxx.A_0008_EJ1859_0000_0017.Channel_12.Output <-> Channel 12/Output
//     PlcTask Outputs/GVL_iXlinker.EtherCAT_Master_EJxxxx.Beckhoff_EJ1xxx.A_0008_EJ1859_0000_0017.Channel_13.Output <-> Channel 13/Output
//     PlcTask Outputs/GVL_iXlinker.EtherCAT_Master_EJxxxx.Beckhoff_EJ1xxx.A_0008_EJ1859_0000_0017.Channel_14.Output <-> Channel 14/Output
//     PlcTask Outputs/GVL_iXlinker.EtherCAT_Master_EJxxxx.Beckhoff_EJ1xxx.A_0008_EJ1859_0000_0017.Channel_15.Output <-> Channel 15/Output
//     PlcTask Outputs/GVL_iXlinker.EtherCAT_Master_EJxxxx.Beckhoff_EJ1xxx.A_0008_EJ1859_0000_0017.Channel_16.Output <-> Channel 16/Output
//     PlcTask Inputs/GVL_iXlinker.EtherCAT_Master_EJxxxx.Beckhoff_EJ1xxx.A_0008_EJ1859_0000_0017.WcState.WcState <-> WcState/WcState
//     PlcTask Inputs/GVL_iXlinker.EtherCAT_Master_EJxxxx.Beckhoff_EJ1xxx.A_0008_EJ1859_0000_0017.WcState.InputToggle <-> WcState/InputToggle
//     PlcTask Inputs/GVL_iXlinker.EtherCAT_Master_EJxxxx.Beckhoff_EJ1xxx.A_0008_EJ1859_0000_0017.InfoData.State <-> InfoData/State
//   PLC/PLC Instance <-> EtherCAT Master EJxxxx/Beckhoff EJ1xxx/A_0009(EJ1889-0000-0017)
//     PlcTask Inputs/GVL_iXlinker.EtherCAT_Master_EJxxxx.Beckhoff_EJ1xxx.A_0009_EJ1889_0000_0017.Channel_1.Input <-> Channel 1/Input
//     PlcTask Inputs/GVL_iXlinker.EtherCAT_Master_EJxxxx.Beckhoff_EJ1xxx.A_0009_EJ1889_0000_0017.Channel_2.Input <-> Channel 2/Input
//     PlcTask Inputs/GVL_iXlinker.EtherCAT_Master_EJxxxx.Beckhoff_EJ1xxx.A_0009_EJ1889_0000_0017.Channel_3.Input <-> Channel 3/Input
//     PlcTask Inputs/GVL_iXlinker.EtherCAT_Master_EJxxxx.Beckhoff_EJ1xxx.A_0009_EJ1889_0000_0017.Channel_4.Input <-> Channel 4/Input
//     PlcTask Inputs/GVL_iXlinker.EtherCAT_Master_EJxxxx.Beckhoff_EJ1xxx.A_0009_EJ1889_0000_0017.Channel_5.Input <-> Channel 5/Input
//     PlcTask Inputs/GVL_iXlinker.EtherCAT_Master_EJxxxx.Beckhoff_EJ1xxx.A_0009_EJ1889_0000_0017.Channel_6.Input <-> Channel 6/Input
//     PlcTask Inputs/GVL_iXlinker.EtherCAT_Master_EJxxxx.Beckhoff_EJ1xxx.A_0009_EJ1889_0000_0017.Channel_7.Input <-> Channel 7/Input
//     PlcTask Inputs/GVL_iXlinker.EtherCAT_Master_EJxxxx.Beckhoff_EJ1xxx.A_0009_EJ1889_0000_0017.Channel_8.Input <-> Channel 8/Input
//     PlcTask Inputs/GVL_iXlinker.EtherCAT_Master_EJxxxx.Beckhoff_EJ1xxx.A_0009_EJ1889_0000_0017.Channel_9.Input <-> Channel 9/Input
//     PlcTask Inputs/GVL_iXlinker.EtherCAT_Master_EJxxxx.Beckhoff_EJ1xxx.A_0009_EJ1889_0000_0017.Channel_10.Input <-> Channel 10/Input
//     PlcTask Inputs/GVL_iXlinker.EtherCAT_Master_EJxxxx.Beckhoff_EJ1xxx.A_0009_EJ1889_0000_0017.Channel_11.Input <-> Channel 11/Input
//     PlcTask Inputs/GVL_iXlinker.EtherCAT_Master_EJxxxx.Beckhoff_EJ1xxx.A_0009_EJ1889_0000_0017.Channel_12.Input <-> Channel 12/Input
//     PlcTask Inputs/GVL_iXlinker.EtherCAT_Master_EJxxxx.Beckhoff_EJ1xxx.A_0009_EJ1889_0000_0017.Channel_13.Input <-> Channel 13/Input
//     PlcTask Inputs/GVL_iXlinker.EtherCAT_Master_EJxxxx.Beckhoff_EJ1xxx.A_0009_EJ1889_0000_0017.Channel_14.Input <-> Channel 14/Input
//     PlcTask Inputs/GVL_iXlinker.EtherCAT_Master_EJxxxx.Beckhoff_EJ1xxx.A_0009_EJ1889_0000_0017.Channel_15.Input <-> Channel 15/Input
//     PlcTask Inputs/GVL_iXlinker.EtherCAT_Master_EJxxxx.Beckhoff_EJ1xxx.A_0009_EJ1889_0000_0017.Channel_16.Input <-> Channel 16/Input
//     PlcTask Inputs/GVL_iXlinker.EtherCAT_Master_EJxxxx.Beckhoff_EJ1xxx.A_0009_EJ1889_0000_0017.WcState.WcState <-> WcState/WcState
//     PlcTask Inputs/GVL_iXlinker.EtherCAT_Master_EJxxxx.Beckhoff_EJ1xxx.A_0009_EJ1889_0000_0017.WcState.InputToggle <-> WcState/InputToggle
//     PlcTask Inputs/GVL_iXlinker.EtherCAT_Master_EJxxxx.Beckhoff_EJ1xxx.A_0009_EJ1889_0000_0017.InfoData.State <-> InfoData/State
//   PLC/PLC Instance <-> EtherCAT Master EJxxxx/Beckhoff EJ1xxx/A_0003(EJ1122-0000-0016)
//     PlcTask Inputs/GVL_iXlinker.EtherCAT_Master_EJxxxx.Beckhoff_EJ1xxx.A_0003_EJ1122_0000_0016.InfoData.State <-> InfoData/State
//   PLC/PLC Instance <-> EtherCAT Master EJxxxx/Beckhoff EJ2xxx
//     PlcTask Inputs/GVL_iXlinker.EtherCAT_Master_EJxxxx.Beckhoff_EJ2xxx.InfoData.State <-> InfoData/State
//   PLC/PLC Instance <-> EtherCAT Master EJxxxx/Beckhoff EJ2xxx/Beckhoff EJ2xxxEK1122
//     PlcTask Inputs/GVL_iXlinker.EtherCAT_Master_EJxxxx.Beckhoff_EJ2xxx.Beckhoff_EJ2xxxEK1122.InfoData.State <-> InfoData/State
//   PLC/PLC Instance <-> EtherCAT Master EJxxxx/Beckhoff EJ2xxx/Beckhoff EJ2xxxEK1122/Beckhoff EJ2xxxsub EK1100
//     PlcTask Inputs/GVL_iXlinker.EtherCAT_Master_EJxxxx.Beckhoff_EJ2xxx.Beckhoff_EJ2xxxEK1122.Beckhoff_EJ2xxxsub_EK1100.InfoData.State <-> InfoData/State
//   PLC/PLC Instance <-> EtherCAT Master EJxxxx/Beckhoff EJ2xxx/A_0001(EJ2008-0000-0017)
//     PlcTask Outputs/GVL_iXlinker.EtherCAT_Master_EJxxxx.Beckhoff_EJ2xxx.A_0001_EJ2008_0000_0017.Channel_1.Output <-> Channel 1/Output
//     PlcTask Outputs/GVL_iXlinker.EtherCAT_Master_EJxxxx.Beckhoff_EJ2xxx.A_0001_EJ2008_0000_0017.Channel_2.Output <-> Channel 2/Output
//     PlcTask Outputs/GVL_iXlinker.EtherCAT_Master_EJxxxx.Beckhoff_EJ2xxx.A_0001_EJ2008_0000_0017.Channel_3.Output <-> Channel 3/Output
//     PlcTask Outputs/GVL_iXlinker.EtherCAT_Master_EJxxxx.Beckhoff_EJ2xxx.A_0001_EJ2008_0000_0017.Channel_4.Output <-> Channel 4/Output
//     PlcTask Outputs/GVL_iXlinker.EtherCAT_Master_EJxxxx.Beckhoff_EJ2xxx.A_0001_EJ2008_0000_0017.Channel_5.Output <-> Channel 5/Output
//     PlcTask Outputs/GVL_iXlinker.EtherCAT_Master_EJxxxx.Beckhoff_EJ2xxx.A_0001_EJ2008_0000_0017.Channel_6.Output <-> Channel 6/Output
//     PlcTask Outputs/GVL_iXlinker.EtherCAT_Master_EJxxxx.Beckhoff_EJ2xxx.A_0001_EJ2008_0000_0017.Channel_7.Output <-> Channel 7/Output
//     PlcTask Outputs/GVL_iXlinker.EtherCAT_Master_EJxxxx.Beckhoff_EJ2xxx.A_0001_EJ2008_0000_0017.Channel_8.Output <-> Channel 8/Output
//     PlcTask Inputs/GVL_iXlinker.EtherCAT_Master_EJxxxx.Beckhoff_EJ2xxx.A_0001_EJ2008_0000_0017.WcState.WcState <-> WcState/WcState
//     PlcTask Inputs/GVL_iXlinker.EtherCAT_Master_EJxxxx.Beckhoff_EJ2xxx.A_0001_EJ2008_0000_0017.InfoData.State <-> InfoData/State
//   PLC/PLC Instance <-> EtherCAT Master EJxxxx/Beckhoff EJ2xxx/A_0002(EJ2008-0000-0018)
//     PlcTask Outputs/GVL_iXlinker.EtherCAT_Master_EJxxxx.Beckhoff_EJ2xxx.A_0002_EJ2008_0000_0018.Channel_1.Output <-> Channel 1/Output
//     PlcTask Outputs/GVL_iXlinker.EtherCAT_Master_EJxxxx.Beckhoff_EJ2xxx.A_0002_EJ2008_0000_0018.Channel_2.Output <-> Channel 2/Output
//     PlcTask Outputs/GVL_iXlinker.EtherCAT_Master_EJxxxx.Beckhoff_EJ2xxx.A_0002_EJ2008_0000_0018.Channel_3.Output <-> Channel 3/Output
//     PlcTask Outputs/GVL_iXlinker.EtherCAT_Master_EJxxxx.Beckhoff_EJ2xxx.A_0002_EJ2008_0000_0018.Channel_4.Output <-> Channel 4/Output
//     PlcTask Outputs/GVL_iXlinker.EtherCAT_Master_EJxxxx.Beckhoff_EJ2xxx.A_0002_EJ2008_0000_0018.Channel_5.Output <-> Channel 5/Output
//     PlcTask Outputs/GVL_iXlinker.EtherCAT_Master_EJxxxx.Beckhoff_EJ2xxx.A_0002_EJ2008_0000_0018.Channel_6.Output <-> Channel 6/Output
//     PlcTask Outputs/GVL_iXlinker.EtherCAT_Master_EJxxxx.Beckhoff_EJ2xxx.A_0002_EJ2008_0000_0018.Channel_7.Output <-> Channel 7/Output
//     PlcTask Outputs/GVL_iXlinker.EtherCAT_Master_EJxxxx.Beckhoff_EJ2xxx.A_0002_EJ2008_0000_0018.Channel_8.Output <-> Channel 8/Output
//     PlcTask Inputs/GVL_iXlinker.EtherCAT_Master_EJxxxx.Beckhoff_EJ2xxx.A_0002_EJ2008_0000_0018.WcState.WcState <-> WcState/WcState
//     PlcTask Inputs/GVL_iXlinker.EtherCAT_Master_EJxxxx.Beckhoff_EJ2xxx.A_0002_EJ2008_0000_0018.InfoData.State <-> InfoData/State
//   PLC/PLC Instance <-> EtherCAT Master EJxxxx/Beckhoff EJ2xxx/A_0003(EJ2128-0000-0016)
//     PlcTask Outputs/GVL_iXlinker.EtherCAT_Master_EJxxxx.Beckhoff_EJ2xxx.A_0003_EJ2128_0000_0016.Channel_1.Output <-> Channel 1/Output
//     PlcTask Outputs/GVL_iXlinker.EtherCAT_Master_EJxxxx.Beckhoff_EJ2xxx.A_0003_EJ2128_0000_0016.Channel_2.Output <-> Channel 2/Output
//     PlcTask Outputs/GVL_iXlinker.EtherCAT_Master_EJxxxx.Beckhoff_EJ2xxx.A_0003_EJ2128_0000_0016.Channel_3.Output <-> Channel 3/Output
//     PlcTask Outputs/GVL_iXlinker.EtherCAT_Master_EJxxxx.Beckhoff_EJ2xxx.A_0003_EJ2128_0000_0016.Channel_4.Output <-> Channel 4/Output
//     PlcTask Outputs/GVL_iXlinker.EtherCAT_Master_EJxxxx.Beckhoff_EJ2xxx.A_0003_EJ2128_0000_0016.Channel_5.Output <-> Channel 5/Output
//     PlcTask Outputs/GVL_iXlinker.EtherCAT_Master_EJxxxx.Beckhoff_EJ2xxx.A_0003_EJ2128_0000_0016.Channel_6.Output <-> Channel 6/Output
//     PlcTask Outputs/GVL_iXlinker.EtherCAT_Master_EJxxxx.Beckhoff_EJ2xxx.A_0003_EJ2128_0000_0016.Channel_7.Output <-> Channel 7/Output
//     PlcTask Outputs/GVL_iXlinker.EtherCAT_Master_EJxxxx.Beckhoff_EJ2xxx.A_0003_EJ2128_0000_0016.Channel_8.Output <-> Channel 8/Output
//     PlcTask Inputs/GVL_iXlinker.EtherCAT_Master_EJxxxx.Beckhoff_EJ2xxx.A_0003_EJ2128_0000_0016.WcState.WcState <-> WcState/WcState
//     PlcTask Inputs/GVL_iXlinker.EtherCAT_Master_EJxxxx.Beckhoff_EJ2xxx.A_0003_EJ2128_0000_0016.InfoData.State <-> InfoData/State
//   PLC/PLC Instance <-> EtherCAT Master EJxxxx/Beckhoff EJ2xxx/A_0004(EJ2502-0000-0023)
//     PlcTask Outputs/GVL_iXlinker.EtherCAT_Master_EJxxxx.Beckhoff_EJ2xxx.A_0004_EJ2502_0000_0023.PWM_Outputs_Channel_1.PWM_output <-> PWM Outputs Channel 1/PWM output
//     PlcTask Outputs/GVL_iXlinker.EtherCAT_Master_EJxxxx.Beckhoff_EJ2xxx.A_0004_EJ2502_0000_0023.PWM_Outputs_Channel_2.PWM_output <-> PWM Outputs Channel 2/PWM output
//     PlcTask Inputs/GVL_iXlinker.EtherCAT_Master_EJxxxx.Beckhoff_EJ2xxx.A_0004_EJ2502_0000_0023.WcState.WcState <-> WcState/WcState
//     PlcTask Inputs/GVL_iXlinker.EtherCAT_Master_EJxxxx.Beckhoff_EJ2xxx.A_0004_EJ2502_0000_0023.InfoData.AdsAddr <-> InfoData/AdsAddr
//     PlcTask Inputs/GVL_iXlinker.EtherCAT_Master_EJxxxx.Beckhoff_EJ2xxx.A_0004_EJ2502_0000_0023.InfoData.State <-> InfoData/State
//   PLC/PLC Instance <-> EtherCAT Master EJxxxx/Beckhoff EJ2xxx/A_0005(EJ2502-0000-0024)
//     PlcTask Outputs/GVL_iXlinker.EtherCAT_Master_EJxxxx.Beckhoff_EJ2xxx.A_0005_EJ2502_0000_0024.PWM_Outputs_Channel_1.PWM_output <-> PWM Outputs Channel 1/PWM output
//     PlcTask Outputs/GVL_iXlinker.EtherCAT_Master_EJxxxx.Beckhoff_EJ2xxx.A_0005_EJ2502_0000_0024.PWM_Outputs_Channel_2.PWM_output <-> PWM Outputs Channel 2/PWM output
//     PlcTask Inputs/GVL_iXlinker.EtherCAT_Master_EJxxxx.Beckhoff_EJ2xxx.A_0005_EJ2502_0000_0024.WcState.WcState <-> WcState/WcState
//     PlcTask Inputs/GVL_iXlinker.EtherCAT_Master_EJxxxx.Beckhoff_EJ2xxx.A_0005_EJ2502_0000_0024.InfoData.AdsAddr <-> InfoData/AdsAddr
//     PlcTask Inputs/GVL_iXlinker.EtherCAT_Master_EJxxxx.Beckhoff_EJ2xxx.A_0005_EJ2502_0000_0024.InfoData.State <-> InfoData/State
//   PLC/PLC Instance <-> EtherCAT Master EJxxxx/Beckhoff EJ2xxx/A_0006(EJ2521-0224-0016)
//     PlcTask Inputs/GVL_iXlinker.EtherCAT_Master_EJxxxx.Beckhoff_EJ2xxx.A_0006_EJ2521_0224_0016.PTO_Status.Status/Sel_Ack_End_counter <-> PTO Status/Status/Sel. Ack/End counter
//     PlcTask Inputs/GVL_iXlinker.EtherCAT_Master_EJxxxx.Beckhoff_EJ2xxx.A_0006_EJ2521_0224_0016.PTO_Status.Status/Ramp_active <-> PTO Status/Status/Ramp active
//     PlcTask Inputs/GVL_iXlinker.EtherCAT_Master_EJxxxx.Beckhoff_EJ2xxx.A_0006_EJ2521_0224_0016.PTO_Status.Status/Error <-> PTO Status/Status/Error
//     PlcTask Inputs/GVL_iXlinker.EtherCAT_Master_EJxxxx.Beckhoff_EJ2xxx.A_0006_EJ2521_0224_0016.PTO_Status.Status/Sync_error <-> PTO Status/Status/Sync error
//     PlcTask Inputs/GVL_iXlinker.EtherCAT_Master_EJxxxx.Beckhoff_EJ2xxx.A_0006_EJ2521_0224_0016.PTO_Status.Status/TxPDO_Toggle <-> PTO Status/Status/TxPDO Toggle
//     PlcTask Inputs/GVL_iXlinker.EtherCAT_Master_EJxxxx.Beckhoff_EJ2xxx.A_0006_EJ2521_0224_0016.ENC_Status_compact.Status/Latch_extern_valid <-> ENC Status compact/Status/Latch extern valid
//     PlcTask Inputs/GVL_iXlinker.EtherCAT_Master_EJxxxx.Beckhoff_EJ2xxx.A_0006_EJ2521_0224_0016.ENC_Status_compact.Status/Set_counter_done <-> ENC Status compact/Status/Set counter done
//     PlcTask Inputs/GVL_iXlinker.EtherCAT_Master_EJxxxx.Beckhoff_EJ2xxx.A_0006_EJ2521_0224_0016.ENC_Status_compact.Status/Counter_underflow <-> ENC Status compact/Status/Counter underflow
//     PlcTask Inputs/GVL_iXlinker.EtherCAT_Master_EJxxxx.Beckhoff_EJ2xxx.A_0006_EJ2521_0224_0016.ENC_Status_compact.Status/Counter_overflow <-> ENC Status compact/Status/Counter overflow
//     PlcTask Inputs/GVL_iXlinker.EtherCAT_Master_EJxxxx.Beckhoff_EJ2xxx.A_0006_EJ2521_0224_0016.ENC_Status_compact.Status/Status_of_extern_latch <-> ENC Status compact/Status/Status of extern latch
//     PlcTask Inputs/GVL_iXlinker.EtherCAT_Master_EJxxxx.Beckhoff_EJ2xxx.A_0006_EJ2521_0224_0016.ENC_Status_compact.Status/Sync_error <-> ENC Status compact/Status/Sync error
//     PlcTask Inputs/GVL_iXlinker.EtherCAT_Master_EJxxxx.Beckhoff_EJ2xxx.A_0006_EJ2521_0224_0016.ENC_Status_compact.Status/TxPDO_Toggle <-> ENC Status compact/Status/TxPDO Toggle
//     PlcTask Inputs/GVL_iXlinker.EtherCAT_Master_EJxxxx.Beckhoff_EJ2xxx.A_0006_EJ2521_0224_0016.ENC_Status_compact.Counter_value <-> ENC Status compact/Counter value
//     PlcTask Inputs/GVL_iXlinker.EtherCAT_Master_EJxxxx.Beckhoff_EJ2xxx.A_0006_EJ2521_0224_0016.ENC_Status_compact.Latch_value <-> ENC Status compact/Latch value
//     PlcTask Inputs/GVL_iXlinker.EtherCAT_Master_EJxxxx.Beckhoff_EJ2xxx.A_0006_EJ2521_0224_0016.PLS_Status_Channel_1.Status/PLS_Enabled <-> PLS Status Channel 1/Status/PLS Enabled
//     PlcTask Inputs/GVL_iXlinker.EtherCAT_Master_EJxxxx.Beckhoff_EJ2xxx.A_0006_EJ2521_0224_0016.PLS_Status_Channel_2.Status/PLS_Enabled <-> PLS Status Channel 2/Status/PLS Enabled
//     PlcTask Inputs/GVL_iXlinker.EtherCAT_Master_EJxxxx.Beckhoff_EJ2xxx.A_0006_EJ2521_0224_0016.PLS_Status_Channel_1.Status/Status_of_output <-> PLS Status Channel 1/Status/Status of output
//     PlcTask Inputs/GVL_iXlinker.EtherCAT_Master_EJxxxx.Beckhoff_EJ2xxx.A_0006_EJ2521_0224_0016.PLS_Status_Channel_2.Status/Status_of_output <-> PLS Status Channel 2/Status/Status of output
//     PlcTask Inputs/GVL_iXlinker.EtherCAT_Master_EJxxxx.Beckhoff_EJ2xxx.A_0006_EJ2521_0224_0016.PLS_Status_Channel_1.Status/Sync_error <-> PLS Status Channel 1/Status/Sync error
//     PlcTask Inputs/GVL_iXlinker.EtherCAT_Master_EJxxxx.Beckhoff_EJ2xxx.A_0006_EJ2521_0224_0016.PLS_Status_Channel_2.Status/Sync_error <-> PLS Status Channel 2/Status/Sync error
//     PlcTask Inputs/GVL_iXlinker.EtherCAT_Master_EJxxxx.Beckhoff_EJ2xxx.A_0006_EJ2521_0224_0016.PLS_Status_Channel_1.Status/TxPDO_Toggle <-> PLS Status Channel 1/Status/TxPDO Toggle
//     PlcTask Inputs/GVL_iXlinker.EtherCAT_Master_EJxxxx.Beckhoff_EJ2xxx.A_0006_EJ2521_0224_0016.PLS_Status_Channel_2.Status/TxPDO_Toggle <-> PLS Status Channel 2/Status/TxPDO Toggle
//     PlcTask Outputs/GVL_iXlinker.EtherCAT_Master_EJxxxx.Beckhoff_EJ2xxx.A_0006_EJ2521_0224_0016.PTO_Control.Control/Frequency_select <-> PTO Control/Control/Frequency select
//     PlcTask Outputs/GVL_iXlinker.EtherCAT_Master_EJxxxx.Beckhoff_EJ2xxx.A_0006_EJ2521_0224_0016.PTO_Control.Control/Disable_ramp <-> PTO Control/Control/Disable ramp
//     PlcTask Outputs/GVL_iXlinker.EtherCAT_Master_EJxxxx.Beckhoff_EJ2xxx.A_0006_EJ2521_0224_0016.PTO_Control.Control/Go_counter <-> PTO Control/Control/Go counter
//     PlcTask Outputs/GVL_iXlinker.EtherCAT_Master_EJxxxx.Beckhoff_EJ2xxx.A_0006_EJ2521_0224_0016.PTO_Control.Frequency_value <-> PTO Control/Frequency value
//     PlcTask Outputs/GVL_iXlinker.EtherCAT_Master_EJxxxx.Beckhoff_EJ2xxx.A_0006_EJ2521_0224_0016.PTO_Target_compact.Target_counter_value <-> PTO Target compact/Target counter value
//     PlcTask Outputs/GVL_iXlinker.EtherCAT_Master_EJxxxx.Beckhoff_EJ2xxx.A_0006_EJ2521_0224_0016.ENC_Control_compact.Control/Enable_latch_extern_on_positive_edge <-> ENC Control compact/Control/Enable latch extern on positive edge
//     PlcTask Outputs/GVL_iXlinker.EtherCAT_Master_EJxxxx.Beckhoff_EJ2xxx.A_0006_EJ2521_0224_0016.ENC_Control_compact.Control/Set_counter <-> ENC Control compact/Control/Set counter
//     PlcTask Outputs/GVL_iXlinker.EtherCAT_Master_EJxxxx.Beckhoff_EJ2xxx.A_0006_EJ2521_0224_0016.ENC_Control_compact.Control/Enable_latch_extern_on_negative_edge <-> ENC Control compact/Control/Enable latch extern on negative edge
//     PlcTask Outputs/GVL_iXlinker.EtherCAT_Master_EJxxxx.Beckhoff_EJ2xxx.A_0006_EJ2521_0224_0016.ENC_Control_compact.Set_counter_value <-> ENC Control compact/Set counter value
//     PlcTask Outputs/GVL_iXlinker.EtherCAT_Master_EJxxxx.Beckhoff_EJ2xxx.A_0006_EJ2521_0224_0016.PLS_Control_compact_Channel_1.Control/Enable_PLS <-> PLS Control compact Channel 1/Control/Enable PLS
//     PlcTask Outputs/GVL_iXlinker.EtherCAT_Master_EJxxxx.Beckhoff_EJ2xxx.A_0006_EJ2521_0224_0016.PLS_Control_compact_Channel_2.Control/Enable_PLS <-> PLS Control compact Channel 2/Control/Enable PLS
//     PlcTask Outputs/GVL_iXlinker.EtherCAT_Master_EJxxxx.Beckhoff_EJ2xxx.A_0006_EJ2521_0224_0016.PLS_Control_compact_Channel_1.Control/Output <-> PLS Control compact Channel 1/Control/Output
//     PlcTask Outputs/GVL_iXlinker.EtherCAT_Master_EJxxxx.Beckhoff_EJ2xxx.A_0006_EJ2521_0224_0016.PLS_Control_compact_Channel_2.Control/Output <-> PLS Control compact Channel 2/Control/Output
//     PlcTask Outputs/GVL_iXlinker.EtherCAT_Master_EJxxxx.Beckhoff_EJ2xxx.A_0006_EJ2521_0224_0016.PLS_Control_compact_Channel_1.Switch_on_value <-> PLS Control compact Channel 1/Switch on value
//     PlcTask Outputs/GVL_iXlinker.EtherCAT_Master_EJxxxx.Beckhoff_EJ2xxx.A_0006_EJ2521_0224_0016.PLS_Control_compact_Channel_2.Switch_on_value <-> PLS Control compact Channel 2/Switch on value
//     PlcTask Outputs/GVL_iXlinker.EtherCAT_Master_EJxxxx.Beckhoff_EJ2xxx.A_0006_EJ2521_0224_0016.PLS_Control_compact_Channel_1.Switch_off_value <-> PLS Control compact Channel 1/Switch off value
//     PlcTask Outputs/GVL_iXlinker.EtherCAT_Master_EJxxxx.Beckhoff_EJ2xxx.A_0006_EJ2521_0224_0016.PLS_Control_compact_Channel_2.Switch_off_value <-> PLS Control compact Channel 2/Switch off value
//     PlcTask Inputs/GVL_iXlinker.EtherCAT_Master_EJxxxx.Beckhoff_EJ2xxx.A_0006_EJ2521_0224_0016.WcState.WcState <-> WcState/WcState
//     PlcTask Inputs/GVL_iXlinker.EtherCAT_Master_EJxxxx.Beckhoff_EJ2xxx.A_0006_EJ2521_0224_0016.WcState.InputToggle <-> WcState/InputToggle
//     PlcTask Inputs/GVL_iXlinker.EtherCAT_Master_EJxxxx.Beckhoff_EJ2xxx.A_0006_EJ2521_0224_0016.InfoData.AdsAddr <-> InfoData/AdsAddr
//     PlcTask Inputs/GVL_iXlinker.EtherCAT_Master_EJxxxx.Beckhoff_EJ2xxx.A_0006_EJ2521_0224_0016.InfoData.State <-> InfoData/State
//   PLC/PLC Instance <-> EtherCAT Master EJxxxx/Beckhoff EJ2xxx/A_0007(EJ2522-0000-0022)
//     PlcTask Inputs/GVL_iXlinker.EtherCAT_Master_EJxxxx.Beckhoff_EJ2xxx.A_0007_EJ2522_0000_0022.PTO_Status_Channel_1.Status/Sel_Ack_End_counter <-> PTO Status Channel 1/Status/Sel. Ack/End counter
//     PlcTask Inputs/GVL_iXlinker.EtherCAT_Master_EJxxxx.Beckhoff_EJ2xxx.A_0007_EJ2522_0000_0022.PTO_Status_Channel_2.Status/Sel_Ack_End_counter <-> PTO Status Channel 2/Status/Sel. Ack/End counter
//     PlcTask Inputs/GVL_iXlinker.EtherCAT_Master_EJxxxx.Beckhoff_EJ2xxx.A_0007_EJ2522_0000_0022.PTO_Status_Channel_1.Status/Ramp_active <-> PTO Status Channel 1/Status/Ramp active
//     PlcTask Inputs/GVL_iXlinker.EtherCAT_Master_EJxxxx.Beckhoff_EJ2xxx.A_0007_EJ2522_0000_0022.PTO_Status_Channel_2.Status/Ramp_active <-> PTO Status Channel 2/Status/Ramp active
//     PlcTask Inputs/GVL_iXlinker.EtherCAT_Master_EJxxxx.Beckhoff_EJ2xxx.A_0007_EJ2522_0000_0022.PTO_Status_Channel_1.Status/Error <-> PTO Status Channel 1/Status/Error
//     PlcTask Inputs/GVL_iXlinker.EtherCAT_Master_EJxxxx.Beckhoff_EJ2xxx.A_0007_EJ2522_0000_0022.PTO_Status_Channel_2.Status/Error <-> PTO Status Channel 2/Status/Error
//     PlcTask Inputs/GVL_iXlinker.EtherCAT_Master_EJxxxx.Beckhoff_EJ2xxx.A_0007_EJ2522_0000_0022.PTO_Status_Channel_1.Status/Sync_error <-> PTO Status Channel 1/Status/Sync error
//     PlcTask Inputs/GVL_iXlinker.EtherCAT_Master_EJxxxx.Beckhoff_EJ2xxx.A_0007_EJ2522_0000_0022.PTO_Status_Channel_2.Status/Sync_error <-> PTO Status Channel 2/Status/Sync error
//     PlcTask Inputs/GVL_iXlinker.EtherCAT_Master_EJxxxx.Beckhoff_EJ2xxx.A_0007_EJ2522_0000_0022.PTO_Status_Channel_1.Status/TxPDO_Toggle <-> PTO Status Channel 1/Status/TxPDO Toggle
//     PlcTask Inputs/GVL_iXlinker.EtherCAT_Master_EJxxxx.Beckhoff_EJ2xxx.A_0007_EJ2522_0000_0022.PTO_Status_Channel_2.Status/TxPDO_Toggle <-> PTO Status Channel 2/Status/TxPDO Toggle
//     PlcTask Inputs/GVL_iXlinker.EtherCAT_Master_EJxxxx.Beckhoff_EJ2xxx.A_0007_EJ2522_0000_0022.ENC_Status_Channel_1.Status/Set_counter_done <-> ENC Status Channel 1/Status/Set counter done
//     PlcTask Inputs/GVL_iXlinker.EtherCAT_Master_EJxxxx.Beckhoff_EJ2xxx.A_0007_EJ2522_0000_0022.ENC_Status_Channel_2.Status/Set_counter_done <-> ENC Status Channel 2/Status/Set counter done
//     PlcTask Inputs/GVL_iXlinker.EtherCAT_Master_EJxxxx.Beckhoff_EJ2xxx.A_0007_EJ2522_0000_0022.ENC_Status_Channel_1.Status/Counter_underflow <-> ENC Status Channel 1/Status/Counter underflow
//     PlcTask Inputs/GVL_iXlinker.EtherCAT_Master_EJxxxx.Beckhoff_EJ2xxx.A_0007_EJ2522_0000_0022.ENC_Status_Channel_2.Status/Counter_underflow <-> ENC Status Channel 2/Status/Counter underflow
//     PlcTask Inputs/GVL_iXlinker.EtherCAT_Master_EJxxxx.Beckhoff_EJ2xxx.A_0007_EJ2522_0000_0022.ENC_Status_Channel_1.Status/Counter_overflow <-> ENC Status Channel 1/Status/Counter overflow
//     PlcTask Inputs/GVL_iXlinker.EtherCAT_Master_EJxxxx.Beckhoff_EJ2xxx.A_0007_EJ2522_0000_0022.ENC_Status_Channel_2.Status/Counter_overflow <-> ENC Status Channel 2/Status/Counter overflow
//     PlcTask Inputs/GVL_iXlinker.EtherCAT_Master_EJxxxx.Beckhoff_EJ2xxx.A_0007_EJ2522_0000_0022.ENC_Status_Channel_1.Status/Sync_error <-> ENC Status Channel 1/Status/Sync error
//     PlcTask Inputs/GVL_iXlinker.EtherCAT_Master_EJxxxx.Beckhoff_EJ2xxx.A_0007_EJ2522_0000_0022.ENC_Status_Channel_2.Status/Sync_error <-> ENC Status Channel 2/Status/Sync error
//     PlcTask Inputs/GVL_iXlinker.EtherCAT_Master_EJxxxx.Beckhoff_EJ2xxx.A_0007_EJ2522_0000_0022.ENC_Status_Channel_1.Status/TxPDO_State <-> ENC Status Channel 1/Status/TxPDO State
//     PlcTask Inputs/GVL_iXlinker.EtherCAT_Master_EJxxxx.Beckhoff_EJ2xxx.A_0007_EJ2522_0000_0022.ENC_Status_Channel_2.Status/TxPDO_State <-> ENC Status Channel 2/Status/TxPDO State
//     PlcTask Inputs/GVL_iXlinker.EtherCAT_Master_EJxxxx.Beckhoff_EJ2xxx.A_0007_EJ2522_0000_0022.ENC_Status_Channel_1.Status/TxPDO_Toggle <-> ENC Status Channel 1/Status/TxPDO Toggle
//     PlcTask Inputs/GVL_iXlinker.EtherCAT_Master_EJxxxx.Beckhoff_EJ2xxx.A_0007_EJ2522_0000_0022.ENC_Status_Channel_2.Status/TxPDO_Toggle <-> ENC Status Channel 2/Status/TxPDO Toggle
//     PlcTask Inputs/GVL_iXlinker.EtherCAT_Master_EJxxxx.Beckhoff_EJ2xxx.A_0007_EJ2522_0000_0022.ENC_Status_Channel_1.Counter_value <-> ENC Status Channel 1/Counter value
//     PlcTask Inputs/GVL_iXlinker.EtherCAT_Master_EJxxxx.Beckhoff_EJ2xxx.A_0007_EJ2522_0000_0022.ENC_Status_Channel_2.Counter_value <-> ENC Status Channel 2/Counter value
//     PlcTask Outputs/GVL_iXlinker.EtherCAT_Master_EJxxxx.Beckhoff_EJ2xxx.A_0007_EJ2522_0000_0022.PTO_Control_Channel_1.Control/Frequency_select <-> PTO Control Channel 1/Control/Frequency select
//     PlcTask Outputs/GVL_iXlinker.EtherCAT_Master_EJxxxx.Beckhoff_EJ2xxx.A_0007_EJ2522_0000_0022.PTO_Control_Channel_2.Control/Frequency_select <-> PTO Control Channel 2/Control/Frequency select
//     PlcTask Outputs/GVL_iXlinker.EtherCAT_Master_EJxxxx.Beckhoff_EJ2xxx.A_0007_EJ2522_0000_0022.PTO_Control_Channel_1.Control/Disable_ramp <-> PTO Control Channel 1/Control/Disable ramp
//     PlcTask Outputs/GVL_iXlinker.EtherCAT_Master_EJxxxx.Beckhoff_EJ2xxx.A_0007_EJ2522_0000_0022.PTO_Control_Channel_2.Control/Disable_ramp <-> PTO Control Channel 2/Control/Disable ramp
//     PlcTask Outputs/GVL_iXlinker.EtherCAT_Master_EJxxxx.Beckhoff_EJ2xxx.A_0007_EJ2522_0000_0022.PTO_Control_Channel_1.Control/Go_counter <-> PTO Control Channel 1/Control/Go counter
//     PlcTask Outputs/GVL_iXlinker.EtherCAT_Master_EJxxxx.Beckhoff_EJ2xxx.A_0007_EJ2522_0000_0022.PTO_Control_Channel_2.Control/Go_counter <-> PTO Control Channel 2/Control/Go counter
//     PlcTask Outputs/GVL_iXlinker.EtherCAT_Master_EJxxxx.Beckhoff_EJ2xxx.A_0007_EJ2522_0000_0022.PTO_Control_Channel_1.Frequency_value <-> PTO Control Channel 1/Frequency value
//     PlcTask Outputs/GVL_iXlinker.EtherCAT_Master_EJxxxx.Beckhoff_EJ2xxx.A_0007_EJ2522_0000_0022.PTO_Control_Channel_2.Frequency_value <-> PTO Control Channel 2/Frequency value
//     PlcTask Outputs/GVL_iXlinker.EtherCAT_Master_EJxxxx.Beckhoff_EJ2xxx.A_0007_EJ2522_0000_0022.PTO_Target_Channel_1.Target_counter_value <-> PTO Target Channel 1/Target counter value
//     PlcTask Outputs/GVL_iXlinker.EtherCAT_Master_EJxxxx.Beckhoff_EJ2xxx.A_0007_EJ2522_0000_0022.PTO_Target_Channel_2.Target_counter_value <-> PTO Target Channel 2/Target counter value
//     PlcTask Outputs/GVL_iXlinker.EtherCAT_Master_EJxxxx.Beckhoff_EJ2xxx.A_0007_EJ2522_0000_0022.ENC_Control_Channel_1.Control/Set_counter <-> ENC Control Channel 1/Control/Set counter
//     PlcTask Outputs/GVL_iXlinker.EtherCAT_Master_EJxxxx.Beckhoff_EJ2xxx.A_0007_EJ2522_0000_0022.ENC_Control_Channel_2.Control/Set_counter <-> ENC Control Channel 2/Control/Set counter
//     PlcTask Outputs/GVL_iXlinker.EtherCAT_Master_EJxxxx.Beckhoff_EJ2xxx.A_0007_EJ2522_0000_0022.ENC_Control_Channel_1.Control/Reserved <-> ENC Control Channel 1/Control/Reserved
//     PlcTask Outputs/GVL_iXlinker.EtherCAT_Master_EJxxxx.Beckhoff_EJ2xxx.A_0007_EJ2522_0000_0022.ENC_Control_Channel_2.Control/Reserved <-> ENC Control Channel 2/Control/Reserved
//     PlcTask Outputs/GVL_iXlinker.EtherCAT_Master_EJxxxx.Beckhoff_EJ2xxx.A_0007_EJ2522_0000_0022.ENC_Control_Channel_1.Set_counter_value <-> ENC Control Channel 1/Set counter value
//     PlcTask Outputs/GVL_iXlinker.EtherCAT_Master_EJxxxx.Beckhoff_EJ2xxx.A_0007_EJ2522_0000_0022.ENC_Control_Channel_2.Set_counter_value <-> ENC Control Channel 2/Set counter value
//     PlcTask Inputs/GVL_iXlinker.EtherCAT_Master_EJxxxx.Beckhoff_EJ2xxx.A_0007_EJ2522_0000_0022.WcState.WcState <-> WcState/WcState
//     PlcTask Inputs/GVL_iXlinker.EtherCAT_Master_EJxxxx.Beckhoff_EJ2xxx.A_0007_EJ2522_0000_0022.WcState.InputToggle <-> WcState/InputToggle
//     PlcTask Inputs/GVL_iXlinker.EtherCAT_Master_EJxxxx.Beckhoff_EJ2xxx.A_0007_EJ2522_0000_0022.InfoData.AdsAddr <-> InfoData/AdsAddr
//     PlcTask Inputs/GVL_iXlinker.EtherCAT_Master_EJxxxx.Beckhoff_EJ2xxx.A_0007_EJ2522_0000_0022.InfoData.State <-> InfoData/State
//   PLC/PLC Instance <-> EtherCAT Master EJxxxx/Beckhoff EJ2xxx/A_0008(EJ2809-0000-0017)
//     PlcTask Outputs/GVL_iXlinker.EtherCAT_Master_EJxxxx.Beckhoff_EJ2xxx.A_0008_EJ2809_0000_0017.Channel_1.Output <-> Channel 1/Output
//     PlcTask Outputs/GVL_iXlinker.EtherCAT_Master_EJxxxx.Beckhoff_EJ2xxx.A_0008_EJ2809_0000_0017.Channel_2.Output <-> Channel 2/Output
//     PlcTask Outputs/GVL_iXlinker.EtherCAT_Master_EJxxxx.Beckhoff_EJ2xxx.A_0008_EJ2809_0000_0017.Channel_3.Output <-> Channel 3/Output
//     PlcTask Outputs/GVL_iXlinker.EtherCAT_Master_EJxxxx.Beckhoff_EJ2xxx.A_0008_EJ2809_0000_0017.Channel_4.Output <-> Channel 4/Output
//     PlcTask Outputs/GVL_iXlinker.EtherCAT_Master_EJxxxx.Beckhoff_EJ2xxx.A_0008_EJ2809_0000_0017.Channel_5.Output <-> Channel 5/Output
//     PlcTask Outputs/GVL_iXlinker.EtherCAT_Master_EJxxxx.Beckhoff_EJ2xxx.A_0008_EJ2809_0000_0017.Channel_6.Output <-> Channel 6/Output
//     PlcTask Outputs/GVL_iXlinker.EtherCAT_Master_EJxxxx.Beckhoff_EJ2xxx.A_0008_EJ2809_0000_0017.Channel_7.Output <-> Channel 7/Output
//     PlcTask Outputs/GVL_iXlinker.EtherCAT_Master_EJxxxx.Beckhoff_EJ2xxx.A_0008_EJ2809_0000_0017.Channel_8.Output <-> Channel 8/Output
//     PlcTask Outputs/GVL_iXlinker.EtherCAT_Master_EJxxxx.Beckhoff_EJ2xxx.A_0008_EJ2809_0000_0017.Channel_9.Output <-> Channel 9/Output
//     PlcTask Outputs/GVL_iXlinker.EtherCAT_Master_EJxxxx.Beckhoff_EJ2xxx.A_0008_EJ2809_0000_0017.Channel_10.Output <-> Channel 10/Output
//     PlcTask Outputs/GVL_iXlinker.EtherCAT_Master_EJxxxx.Beckhoff_EJ2xxx.A_0008_EJ2809_0000_0017.Channel_11.Output <-> Channel 11/Output
//     PlcTask Outputs/GVL_iXlinker.EtherCAT_Master_EJxxxx.Beckhoff_EJ2xxx.A_0008_EJ2809_0000_0017.Channel_12.Output <-> Channel 12/Output
//     PlcTask Outputs/GVL_iXlinker.EtherCAT_Master_EJxxxx.Beckhoff_EJ2xxx.A_0008_EJ2809_0000_0017.Channel_13.Output <-> Channel 13/Output
//     PlcTask Outputs/GVL_iXlinker.EtherCAT_Master_EJxxxx.Beckhoff_EJ2xxx.A_0008_EJ2809_0000_0017.Channel_14.Output <-> Channel 14/Output
//     PlcTask Outputs/GVL_iXlinker.EtherCAT_Master_EJxxxx.Beckhoff_EJ2xxx.A_0008_EJ2809_0000_0017.Channel_15.Output <-> Channel 15/Output
//     PlcTask Outputs/GVL_iXlinker.EtherCAT_Master_EJxxxx.Beckhoff_EJ2xxx.A_0008_EJ2809_0000_0017.Channel_16.Output <-> Channel 16/Output
//     PlcTask Inputs/GVL_iXlinker.EtherCAT_Master_EJxxxx.Beckhoff_EJ2xxx.A_0008_EJ2809_0000_0017.WcState.WcState <-> WcState/WcState
//     PlcTask Inputs/GVL_iXlinker.EtherCAT_Master_EJxxxx.Beckhoff_EJ2xxx.A_0008_EJ2809_0000_0017.InfoData.State <-> InfoData/State
//   PLC/PLC Instance <-> EtherCAT Master EJxxxx/Beckhoff EJ2xxx/A_0009(EJ2889-0000-0016)
//     PlcTask Outputs/GVL_iXlinker.EtherCAT_Master_EJxxxx.Beckhoff_EJ2xxx.A_0009_EJ2889_0000_0016.Channel_1.Output <-> Channel 1/Output
//     PlcTask Outputs/GVL_iXlinker.EtherCAT_Master_EJxxxx.Beckhoff_EJ2xxx.A_0009_EJ2889_0000_0016.Channel_2.Output <-> Channel 2/Output
//     PlcTask Outputs/GVL_iXlinker.EtherCAT_Master_EJxxxx.Beckhoff_EJ2xxx.A_0009_EJ2889_0000_0016.Channel_3.Output <-> Channel 3/Output
//     PlcTask Outputs/GVL_iXlinker.EtherCAT_Master_EJxxxx.Beckhoff_EJ2xxx.A_0009_EJ2889_0000_0016.Channel_4.Output <-> Channel 4/Output
//     PlcTask Outputs/GVL_iXlinker.EtherCAT_Master_EJxxxx.Beckhoff_EJ2xxx.A_0009_EJ2889_0000_0016.Channel_5.Output <-> Channel 5/Output
//     PlcTask Outputs/GVL_iXlinker.EtherCAT_Master_EJxxxx.Beckhoff_EJ2xxx.A_0009_EJ2889_0000_0016.Channel_6.Output <-> Channel 6/Output
//     PlcTask Outputs/GVL_iXlinker.EtherCAT_Master_EJxxxx.Beckhoff_EJ2xxx.A_0009_EJ2889_0000_0016.Channel_7.Output <-> Channel 7/Output
//     PlcTask Outputs/GVL_iXlinker.EtherCAT_Master_EJxxxx.Beckhoff_EJ2xxx.A_0009_EJ2889_0000_0016.Channel_8.Output <-> Channel 8/Output
//     PlcTask Outputs/GVL_iXlinker.EtherCAT_Master_EJxxxx.Beckhoff_EJ2xxx.A_0009_EJ2889_0000_0016.Channel_9.Output <-> Channel 9/Output
//     PlcTask Outputs/GVL_iXlinker.EtherCAT_Master_EJxxxx.Beckhoff_EJ2xxx.A_0009_EJ2889_0000_0016.Channel_10.Output <-> Channel 10/Output
//     PlcTask Outputs/GVL_iXlinker.EtherCAT_Master_EJxxxx.Beckhoff_EJ2xxx.A_0009_EJ2889_0000_0016.Channel_11.Output <-> Channel 11/Output
//     PlcTask Outputs/GVL_iXlinker.EtherCAT_Master_EJxxxx.Beckhoff_EJ2xxx.A_0009_EJ2889_0000_0016.Channel_12.Output <-> Channel 12/Output
//     PlcTask Outputs/GVL_iXlinker.EtherCAT_Master_EJxxxx.Beckhoff_EJ2xxx.A_0009_EJ2889_0000_0016.Channel_13.Output <-> Channel 13/Output
//     PlcTask Outputs/GVL_iXlinker.EtherCAT_Master_EJxxxx.Beckhoff_EJ2xxx.A_0009_EJ2889_0000_0016.Channel_14.Output <-> Channel 14/Output
//     PlcTask Outputs/GVL_iXlinker.EtherCAT_Master_EJxxxx.Beckhoff_EJ2xxx.A_0009_EJ2889_0000_0016.Channel_15.Output <-> Channel 15/Output
//     PlcTask Outputs/GVL_iXlinker.EtherCAT_Master_EJxxxx.Beckhoff_EJ2xxx.A_0009_EJ2889_0000_0016.Channel_16.Output <-> Channel 16/Output
//     PlcTask Inputs/GVL_iXlinker.EtherCAT_Master_EJxxxx.Beckhoff_EJ2xxx.A_0009_EJ2889_0000_0016.WcState.WcState <-> WcState/WcState
//     PlcTask Inputs/GVL_iXlinker.EtherCAT_Master_EJxxxx.Beckhoff_EJ2xxx.A_0009_EJ2889_0000_0016.InfoData.State <-> InfoData/State
//   PLC/PLC Instance <-> EtherCAT Master EJxxxx/Beckhoff EJ2xxx/A_0010(EJ2889-0000-0017)
//     PlcTask Outputs/GVL_iXlinker.EtherCAT_Master_EJxxxx.Beckhoff_EJ2xxx.A_0010_EJ2889_0000_0017.Channel_1.Output <-> Channel 1/Output
//     PlcTask Outputs/GVL_iXlinker.EtherCAT_Master_EJxxxx.Beckhoff_EJ2xxx.A_0010_EJ2889_0000_0017.Channel_2.Output <-> Channel 2/Output
//     PlcTask Outputs/GVL_iXlinker.EtherCAT_Master_EJxxxx.Beckhoff_EJ2xxx.A_0010_EJ2889_0000_0017.Channel_3.Output <-> Channel 3/Output
//     PlcTask Outputs/GVL_iXlinker.EtherCAT_Master_EJxxxx.Beckhoff_EJ2xxx.A_0010_EJ2889_0000_0017.Channel_4.Output <-> Channel 4/Output
//     PlcTask Outputs/GVL_iXlinker.EtherCAT_Master_EJxxxx.Beckhoff_EJ2xxx.A_0010_EJ2889_0000_0017.Channel_5.Output <-> Channel 5/Output
//     PlcTask Outputs/GVL_iXlinker.EtherCAT_Master_EJxxxx.Beckhoff_EJ2xxx.A_0010_EJ2889_0000_0017.Channel_6.Output <-> Channel 6/Output
//     PlcTask Outputs/GVL_iXlinker.EtherCAT_Master_EJxxxx.Beckhoff_EJ2xxx.A_0010_EJ2889_0000_0017.Channel_7.Output <-> Channel 7/Output
//     PlcTask Outputs/GVL_iXlinker.EtherCAT_Master_EJxxxx.Beckhoff_EJ2xxx.A_0010_EJ2889_0000_0017.Channel_8.Output <-> Channel 8/Output
//     PlcTask Outputs/GVL_iXlinker.EtherCAT_Master_EJxxxx.Beckhoff_EJ2xxx.A_0010_EJ2889_0000_0017.Channel_9.Output <-> Channel 9/Output
//     PlcTask Outputs/GVL_iXlinker.EtherCAT_Master_EJxxxx.Beckhoff_EJ2xxx.A_0010_EJ2889_0000_0017.Channel_10.Output <-> Channel 10/Output
//     PlcTask Outputs/GVL_iXlinker.EtherCAT_Master_EJxxxx.Beckhoff_EJ2xxx.A_0010_EJ2889_0000_0017.Channel_11.Output <-> Channel 11/Output
//     PlcTask Outputs/GVL_iXlinker.EtherCAT_Master_EJxxxx.Beckhoff_EJ2xxx.A_0010_EJ2889_0000_0017.Channel_12.Output <-> Channel 12/Output
//     PlcTask Outputs/GVL_iXlinker.EtherCAT_Master_EJxxxx.Beckhoff_EJ2xxx.A_0010_EJ2889_0000_0017.Channel_13.Output <-> Channel 13/Output
//     PlcTask Outputs/GVL_iXlinker.EtherCAT_Master_EJxxxx.Beckhoff_EJ2xxx.A_0010_EJ2889_0000_0017.Channel_14.Output <-> Channel 14/Output
//     PlcTask Outputs/GVL_iXlinker.EtherCAT_Master_EJxxxx.Beckhoff_EJ2xxx.A_0010_EJ2889_0000_0017.Channel_15.Output <-> Channel 15/Output
//     PlcTask Outputs/GVL_iXlinker.EtherCAT_Master_EJxxxx.Beckhoff_EJ2xxx.A_0010_EJ2889_0000_0017.Channel_16.Output <-> Channel 16/Output
//     PlcTask Inputs/GVL_iXlinker.EtherCAT_Master_EJxxxx.Beckhoff_EJ2xxx.A_0010_EJ2889_0000_0017.WcState.WcState <-> WcState/WcState
//     PlcTask Inputs/GVL_iXlinker.EtherCAT_Master_EJxxxx.Beckhoff_EJ2xxx.A_0010_EJ2889_0000_0017.InfoData.State <-> InfoData/State
//   PLC/PLC Instance <-> EtherCAT Master EJxxxx/Beckhoff EJ3xxx
//     PlcTask Inputs/GVL_iXlinker.EtherCAT_Master_EJxxxx.Beckhoff_EJ3xxx.InfoData.State <-> InfoData/State
//   PLC/PLC Instance <-> EtherCAT Master EJxxxx/Beckhoff EJ3xxx/Beckhoff EJ3xxxEK1122
//     PlcTask Inputs/GVL_iXlinker.EtherCAT_Master_EJxxxx.Beckhoff_EJ3xxx.Beckhoff_EJ3xxxEK1122.InfoData.State <-> InfoData/State
//   PLC/PLC Instance <-> EtherCAT Master EJxxxx/Beckhoff EJ3xxx/Beckhoff EJ3xxxEK1122/Beckhoff EJ3xxxsub EK1100
//     PlcTask Inputs/GVL_iXlinker.EtherCAT_Master_EJxxxx.Beckhoff_EJ3xxx.Beckhoff_EJ3xxxEK1122.Beckhoff_EJ3xxxsub_EK1100.InfoData.State <-> InfoData/State
//   PLC/PLC Instance <-> EtherCAT Master EJxxxx/Beckhoff EJ3xxx/A_0001(EJ3004-0000-0019)
//     PlcTask Inputs/GVL_iXlinker.EtherCAT_Master_EJxxxx.Beckhoff_EJ3xxx.A_0001_EJ3004_0000_0019.AI_Standard_Channel_1.Status/Underrange <-> AI Standard Channel 1/Status/Underrange
//     PlcTask Inputs/GVL_iXlinker.EtherCAT_Master_EJxxxx.Beckhoff_EJ3xxx.A_0001_EJ3004_0000_0019.AI_Standard_Channel_2.Status/Underrange <-> AI Standard Channel 2/Status/Underrange
//     PlcTask Inputs/GVL_iXlinker.EtherCAT_Master_EJxxxx.Beckhoff_EJ3xxx.A_0001_EJ3004_0000_0019.AI_Standard_Channel_3.Status/Underrange <-> AI Standard Channel 3/Status/Underrange
//     PlcTask Inputs/GVL_iXlinker.EtherCAT_Master_EJxxxx.Beckhoff_EJ3xxx.A_0001_EJ3004_0000_0019.AI_Standard_Channel_4.Status/Underrange <-> AI Standard Channel 4/Status/Underrange
//     PlcTask Inputs/GVL_iXlinker.EtherCAT_Master_EJxxxx.Beckhoff_EJ3xxx.A_0001_EJ3004_0000_0019.AI_Standard_Channel_1.Status/Overrange <-> AI Standard Channel 1/Status/Overrange
//     PlcTask Inputs/GVL_iXlinker.EtherCAT_Master_EJxxxx.Beckhoff_EJ3xxx.A_0001_EJ3004_0000_0019.AI_Standard_Channel_2.Status/Overrange <-> AI Standard Channel 2/Status/Overrange
//     PlcTask Inputs/GVL_iXlinker.EtherCAT_Master_EJxxxx.Beckhoff_EJ3xxx.A_0001_EJ3004_0000_0019.AI_Standard_Channel_3.Status/Overrange <-> AI Standard Channel 3/Status/Overrange
//     PlcTask Inputs/GVL_iXlinker.EtherCAT_Master_EJxxxx.Beckhoff_EJ3xxx.A_0001_EJ3004_0000_0019.AI_Standard_Channel_4.Status/Overrange <-> AI Standard Channel 4/Status/Overrange
//     PlcTask Inputs/GVL_iXlinker.EtherCAT_Master_EJxxxx.Beckhoff_EJ3xxx.A_0001_EJ3004_0000_0019.AI_Standard_Channel_1.Status/Limit_1 <-> AI Standard Channel 1/Status/Limit 1
//     PlcTask Inputs/GVL_iXlinker.EtherCAT_Master_EJxxxx.Beckhoff_EJ3xxx.A_0001_EJ3004_0000_0019.AI_Standard_Channel_1.Status/Limit_2 <-> AI Standard Channel 1/Status/Limit 2
//     PlcTask Inputs/GVL_iXlinker.EtherCAT_Master_EJxxxx.Beckhoff_EJ3xxx.A_0001_EJ3004_0000_0019.AI_Standard_Channel_2.Status/Limit_1 <-> AI Standard Channel 2/Status/Limit 1
//     PlcTask Inputs/GVL_iXlinker.EtherCAT_Master_EJxxxx.Beckhoff_EJ3xxx.A_0001_EJ3004_0000_0019.AI_Standard_Channel_2.Status/Limit_2 <-> AI Standard Channel 2/Status/Limit 2
//     PlcTask Inputs/GVL_iXlinker.EtherCAT_Master_EJxxxx.Beckhoff_EJ3xxx.A_0001_EJ3004_0000_0019.AI_Standard_Channel_3.Status/Limit_1 <-> AI Standard Channel 3/Status/Limit 1
//     PlcTask Inputs/GVL_iXlinker.EtherCAT_Master_EJxxxx.Beckhoff_EJ3xxx.A_0001_EJ3004_0000_0019.AI_Standard_Channel_3.Status/Limit_2 <-> AI Standard Channel 3/Status/Limit 2
//     PlcTask Inputs/GVL_iXlinker.EtherCAT_Master_EJxxxx.Beckhoff_EJ3xxx.A_0001_EJ3004_0000_0019.AI_Standard_Channel_4.Status/Limit_1 <-> AI Standard Channel 4/Status/Limit 1
//     PlcTask Inputs/GVL_iXlinker.EtherCAT_Master_EJxxxx.Beckhoff_EJ3xxx.A_0001_EJ3004_0000_0019.AI_Standard_Channel_4.Status/Limit_2 <-> AI Standard Channel 4/Status/Limit 2
//     PlcTask Inputs/GVL_iXlinker.EtherCAT_Master_EJxxxx.Beckhoff_EJ3xxx.A_0001_EJ3004_0000_0019.AI_Standard_Channel_1.Status/Error <-> AI Standard Channel 1/Status/Error
//     PlcTask Inputs/GVL_iXlinker.EtherCAT_Master_EJxxxx.Beckhoff_EJ3xxx.A_0001_EJ3004_0000_0019.AI_Standard_Channel_2.Status/Error <-> AI Standard Channel 2/Status/Error
//     PlcTask Inputs/GVL_iXlinker.EtherCAT_Master_EJxxxx.Beckhoff_EJ3xxx.A_0001_EJ3004_0000_0019.AI_Standard_Channel_3.Status/Error <-> AI Standard Channel 3/Status/Error
//     PlcTask Inputs/GVL_iXlinker.EtherCAT_Master_EJxxxx.Beckhoff_EJ3xxx.A_0001_EJ3004_0000_0019.AI_Standard_Channel_4.Status/Error <-> AI Standard Channel 4/Status/Error
//     PlcTask Inputs/GVL_iXlinker.EtherCAT_Master_EJxxxx.Beckhoff_EJ3xxx.A_0001_EJ3004_0000_0019.AI_Standard_Channel_1.Status/TxPDO_State <-> AI Standard Channel 1/Status/TxPDO State
//     PlcTask Inputs/GVL_iXlinker.EtherCAT_Master_EJxxxx.Beckhoff_EJ3xxx.A_0001_EJ3004_0000_0019.AI_Standard_Channel_2.Status/TxPDO_State <-> AI Standard Channel 2/Status/TxPDO State
//     PlcTask Inputs/GVL_iXlinker.EtherCAT_Master_EJxxxx.Beckhoff_EJ3xxx.A_0001_EJ3004_0000_0019.AI_Standard_Channel_3.Status/TxPDO_State <-> AI Standard Channel 3/Status/TxPDO State
//     PlcTask Inputs/GVL_iXlinker.EtherCAT_Master_EJxxxx.Beckhoff_EJ3xxx.A_0001_EJ3004_0000_0019.AI_Standard_Channel_4.Status/TxPDO_State <-> AI Standard Channel 4/Status/TxPDO State
//     PlcTask Inputs/GVL_iXlinker.EtherCAT_Master_EJxxxx.Beckhoff_EJ3xxx.A_0001_EJ3004_0000_0019.AI_Standard_Channel_1.Status/TxPDO_Toggle <-> AI Standard Channel 1/Status/TxPDO Toggle
//     PlcTask Inputs/GVL_iXlinker.EtherCAT_Master_EJxxxx.Beckhoff_EJ3xxx.A_0001_EJ3004_0000_0019.AI_Standard_Channel_2.Status/TxPDO_Toggle <-> AI Standard Channel 2/Status/TxPDO Toggle
//     PlcTask Inputs/GVL_iXlinker.EtherCAT_Master_EJxxxx.Beckhoff_EJ3xxx.A_0001_EJ3004_0000_0019.AI_Standard_Channel_3.Status/TxPDO_Toggle <-> AI Standard Channel 3/Status/TxPDO Toggle
//     PlcTask Inputs/GVL_iXlinker.EtherCAT_Master_EJxxxx.Beckhoff_EJ3xxx.A_0001_EJ3004_0000_0019.AI_Standard_Channel_4.Status/TxPDO_Toggle <-> AI Standard Channel 4/Status/TxPDO Toggle
//     PlcTask Inputs/GVL_iXlinker.EtherCAT_Master_EJxxxx.Beckhoff_EJ3xxx.A_0001_EJ3004_0000_0019.AI_Standard_Channel_1.Value <-> AI Standard Channel 1/Value
//     PlcTask Inputs/GVL_iXlinker.EtherCAT_Master_EJxxxx.Beckhoff_EJ3xxx.A_0001_EJ3004_0000_0019.AI_Standard_Channel_2.Value <-> AI Standard Channel 2/Value
//     PlcTask Inputs/GVL_iXlinker.EtherCAT_Master_EJxxxx.Beckhoff_EJ3xxx.A_0001_EJ3004_0000_0019.AI_Standard_Channel_3.Value <-> AI Standard Channel 3/Value
//     PlcTask Inputs/GVL_iXlinker.EtherCAT_Master_EJxxxx.Beckhoff_EJ3xxx.A_0001_EJ3004_0000_0019.AI_Standard_Channel_4.Value <-> AI Standard Channel 4/Value
//     PlcTask Inputs/GVL_iXlinker.EtherCAT_Master_EJxxxx.Beckhoff_EJ3xxx.A_0001_EJ3004_0000_0019.WcState.WcState <-> WcState/WcState
//     PlcTask Inputs/GVL_iXlinker.EtherCAT_Master_EJxxxx.Beckhoff_EJ3xxx.A_0001_EJ3004_0000_0019.WcState.InputToggle <-> WcState/InputToggle
//     PlcTask Inputs/GVL_iXlinker.EtherCAT_Master_EJxxxx.Beckhoff_EJ3xxx.A_0001_EJ3004_0000_0019.InfoData.AdsAddr <-> InfoData/AdsAddr
//     PlcTask Inputs/GVL_iXlinker.EtherCAT_Master_EJxxxx.Beckhoff_EJ3xxx.A_0001_EJ3004_0000_0019.InfoData.State <-> InfoData/State
//   PLC/PLC Instance <-> EtherCAT Master EJxxxx/Beckhoff EJ3xxx/A_0002(EJ3004-0000-0020)
//     PlcTask Inputs/GVL_iXlinker.EtherCAT_Master_EJxxxx.Beckhoff_EJ3xxx.A_0002_EJ3004_0000_0020.AI_Standard_Channel_1.Status/Underrange <-> AI Standard Channel 1/Status/Underrange
//     PlcTask Inputs/GVL_iXlinker.EtherCAT_Master_EJxxxx.Beckhoff_EJ3xxx.A_0002_EJ3004_0000_0020.AI_Standard_Channel_2.Status/Underrange <-> AI Standard Channel 2/Status/Underrange
//     PlcTask Inputs/GVL_iXlinker.EtherCAT_Master_EJxxxx.Beckhoff_EJ3xxx.A_0002_EJ3004_0000_0020.AI_Standard_Channel_3.Status/Underrange <-> AI Standard Channel 3/Status/Underrange
//     PlcTask Inputs/GVL_iXlinker.EtherCAT_Master_EJxxxx.Beckhoff_EJ3xxx.A_0002_EJ3004_0000_0020.AI_Standard_Channel_4.Status/Underrange <-> AI Standard Channel 4/Status/Underrange
//     PlcTask Inputs/GVL_iXlinker.EtherCAT_Master_EJxxxx.Beckhoff_EJ3xxx.A_0002_EJ3004_0000_0020.AI_Standard_Channel_1.Status/Overrange <-> AI Standard Channel 1/Status/Overrange
//     PlcTask Inputs/GVL_iXlinker.EtherCAT_Master_EJxxxx.Beckhoff_EJ3xxx.A_0002_EJ3004_0000_0020.AI_Standard_Channel_2.Status/Overrange <-> AI Standard Channel 2/Status/Overrange
//     PlcTask Inputs/GVL_iXlinker.EtherCAT_Master_EJxxxx.Beckhoff_EJ3xxx.A_0002_EJ3004_0000_0020.AI_Standard_Channel_3.Status/Overrange <-> AI Standard Channel 3/Status/Overrange
//     PlcTask Inputs/GVL_iXlinker.EtherCAT_Master_EJxxxx.Beckhoff_EJ3xxx.A_0002_EJ3004_0000_0020.AI_Standard_Channel_4.Status/Overrange <-> AI Standard Channel 4/Status/Overrange
//     PlcTask Inputs/GVL_iXlinker.EtherCAT_Master_EJxxxx.Beckhoff_EJ3xxx.A_0002_EJ3004_0000_0020.AI_Standard_Channel_1.Status/Limit_1 <-> AI Standard Channel 1/Status/Limit 1
//     PlcTask Inputs/GVL_iXlinker.EtherCAT_Master_EJxxxx.Beckhoff_EJ3xxx.A_0002_EJ3004_0000_0020.AI_Standard_Channel_1.Status/Limit_2 <-> AI Standard Channel 1/Status/Limit 2
//     PlcTask Inputs/GVL_iXlinker.EtherCAT_Master_EJxxxx.Beckhoff_EJ3xxx.A_0002_EJ3004_0000_0020.AI_Standard_Channel_2.Status/Limit_1 <-> AI Standard Channel 2/Status/Limit 1
//     PlcTask Inputs/GVL_iXlinker.EtherCAT_Master_EJxxxx.Beckhoff_EJ3xxx.A_0002_EJ3004_0000_0020.AI_Standard_Channel_2.Status/Limit_2 <-> AI Standard Channel 2/Status/Limit 2
//     PlcTask Inputs/GVL_iXlinker.EtherCAT_Master_EJxxxx.Beckhoff_EJ3xxx.A_0002_EJ3004_0000_0020.AI_Standard_Channel_3.Status/Limit_1 <-> AI Standard Channel 3/Status/Limit 1
//     PlcTask Inputs/GVL_iXlinker.EtherCAT_Master_EJxxxx.Beckhoff_EJ3xxx.A_0002_EJ3004_0000_0020.AI_Standard_Channel_3.Status/Limit_2 <-> AI Standard Channel 3/Status/Limit 2
//     PlcTask Inputs/GVL_iXlinker.EtherCAT_Master_EJxxxx.Beckhoff_EJ3xxx.A_0002_EJ3004_0000_0020.AI_Standard_Channel_4.Status/Limit_1 <-> AI Standard Channel 4/Status/Limit 1
//     PlcTask Inputs/GVL_iXlinker.EtherCAT_Master_EJxxxx.Beckhoff_EJ3xxx.A_0002_EJ3004_0000_0020.AI_Standard_Channel_4.Status/Limit_2 <-> AI Standard Channel 4/Status/Limit 2
//     PlcTask Inputs/GVL_iXlinker.EtherCAT_Master_EJxxxx.Beckhoff_EJ3xxx.A_0002_EJ3004_0000_0020.AI_Standard_Channel_1.Status/Error <-> AI Standard Channel 1/Status/Error
//     PlcTask Inputs/GVL_iXlinker.EtherCAT_Master_EJxxxx.Beckhoff_EJ3xxx.A_0002_EJ3004_0000_0020.AI_Standard_Channel_2.Status/Error <-> AI Standard Channel 2/Status/Error
//     PlcTask Inputs/GVL_iXlinker.EtherCAT_Master_EJxxxx.Beckhoff_EJ3xxx.A_0002_EJ3004_0000_0020.AI_Standard_Channel_3.Status/Error <-> AI Standard Channel 3/Status/Error
//     PlcTask Inputs/GVL_iXlinker.EtherCAT_Master_EJxxxx.Beckhoff_EJ3xxx.A_0002_EJ3004_0000_0020.AI_Standard_Channel_4.Status/Error <-> AI Standard Channel 4/Status/Error
//     PlcTask Inputs/GVL_iXlinker.EtherCAT_Master_EJxxxx.Beckhoff_EJ3xxx.A_0002_EJ3004_0000_0020.AI_Standard_Channel_1.Status/TxPDO_State <-> AI Standard Channel 1/Status/TxPDO State
//     PlcTask Inputs/GVL_iXlinker.EtherCAT_Master_EJxxxx.Beckhoff_EJ3xxx.A_0002_EJ3004_0000_0020.AI_Standard_Channel_2.Status/TxPDO_State <-> AI Standard Channel 2/Status/TxPDO State
//     PlcTask Inputs/GVL_iXlinker.EtherCAT_Master_EJxxxx.Beckhoff_EJ3xxx.A_0002_EJ3004_0000_0020.AI_Standard_Channel_3.Status/TxPDO_State <-> AI Standard Channel 3/Status/TxPDO State
//     PlcTask Inputs/GVL_iXlinker.EtherCAT_Master_EJxxxx.Beckhoff_EJ3xxx.A_0002_EJ3004_0000_0020.AI_Standard_Channel_4.Status/TxPDO_State <-> AI Standard Channel 4/Status/TxPDO State
//     PlcTask Inputs/GVL_iXlinker.EtherCAT_Master_EJxxxx.Beckhoff_EJ3xxx.A_0002_EJ3004_0000_0020.AI_Standard_Channel_1.Status/TxPDO_Toggle <-> AI Standard Channel 1/Status/TxPDO Toggle
//     PlcTask Inputs/GVL_iXlinker.EtherCAT_Master_EJxxxx.Beckhoff_EJ3xxx.A_0002_EJ3004_0000_0020.AI_Standard_Channel_2.Status/TxPDO_Toggle <-> AI Standard Channel 2/Status/TxPDO Toggle
//     PlcTask Inputs/GVL_iXlinker.EtherCAT_Master_EJxxxx.Beckhoff_EJ3xxx.A_0002_EJ3004_0000_0020.AI_Standard_Channel_3.Status/TxPDO_Toggle <-> AI Standard Channel 3/Status/TxPDO Toggle
//     PlcTask Inputs/GVL_iXlinker.EtherCAT_Master_EJxxxx.Beckhoff_EJ3xxx.A_0002_EJ3004_0000_0020.AI_Standard_Channel_4.Status/TxPDO_Toggle <-> AI Standard Channel 4/Status/TxPDO Toggle
//     PlcTask Inputs/GVL_iXlinker.EtherCAT_Master_EJxxxx.Beckhoff_EJ3xxx.A_0002_EJ3004_0000_0020.AI_Standard_Channel_1.Value <-> AI Standard Channel 1/Value
//     PlcTask Inputs/GVL_iXlinker.EtherCAT_Master_EJxxxx.Beckhoff_EJ3xxx.A_0002_EJ3004_0000_0020.AI_Standard_Channel_2.Value <-> AI Standard Channel 2/Value
//     PlcTask Inputs/GVL_iXlinker.EtherCAT_Master_EJxxxx.Beckhoff_EJ3xxx.A_0002_EJ3004_0000_0020.AI_Standard_Channel_3.Value <-> AI Standard Channel 3/Value
//     PlcTask Inputs/GVL_iXlinker.EtherCAT_Master_EJxxxx.Beckhoff_EJ3xxx.A_0002_EJ3004_0000_0020.AI_Standard_Channel_4.Value <-> AI Standard Channel 4/Value
//     PlcTask Inputs/GVL_iXlinker.EtherCAT_Master_EJxxxx.Beckhoff_EJ3xxx.A_0002_EJ3004_0000_0020.WcState.WcState <-> WcState/WcState
//     PlcTask Inputs/GVL_iXlinker.EtherCAT_Master_EJxxxx.Beckhoff_EJ3xxx.A_0002_EJ3004_0000_0020.WcState.InputToggle <-> WcState/InputToggle
//     PlcTask Inputs/GVL_iXlinker.EtherCAT_Master_EJxxxx.Beckhoff_EJ3xxx.A_0002_EJ3004_0000_0020.InfoData.AdsAddr <-> InfoData/AdsAddr
//     PlcTask Inputs/GVL_iXlinker.EtherCAT_Master_EJxxxx.Beckhoff_EJ3xxx.A_0002_EJ3004_0000_0020.InfoData.State <-> InfoData/State
//   PLC/PLC Instance <-> EtherCAT Master EJxxxx/Beckhoff EJ3xxx/A_0003(EJ3004-0000-0021)
//     PlcTask Inputs/GVL_iXlinker.EtherCAT_Master_EJxxxx.Beckhoff_EJ3xxx.A_0003_EJ3004_0000_0021.AI_Standard_Channel_1.Status/Underrange <-> AI Standard Channel 1/Status/Underrange
//     PlcTask Inputs/GVL_iXlinker.EtherCAT_Master_EJxxxx.Beckhoff_EJ3xxx.A_0003_EJ3004_0000_0021.AI_Standard_Channel_2.Status/Underrange <-> AI Standard Channel 2/Status/Underrange
//     PlcTask Inputs/GVL_iXlinker.EtherCAT_Master_EJxxxx.Beckhoff_EJ3xxx.A_0003_EJ3004_0000_0021.AI_Standard_Channel_3.Status/Underrange <-> AI Standard Channel 3/Status/Underrange
//     PlcTask Inputs/GVL_iXlinker.EtherCAT_Master_EJxxxx.Beckhoff_EJ3xxx.A_0003_EJ3004_0000_0021.AI_Standard_Channel_4.Status/Underrange <-> AI Standard Channel 4/Status/Underrange
//     PlcTask Inputs/GVL_iXlinker.EtherCAT_Master_EJxxxx.Beckhoff_EJ3xxx.A_0003_EJ3004_0000_0021.AI_Standard_Channel_1.Status/Overrange <-> AI Standard Channel 1/Status/Overrange
//     PlcTask Inputs/GVL_iXlinker.EtherCAT_Master_EJxxxx.Beckhoff_EJ3xxx.A_0003_EJ3004_0000_0021.AI_Standard_Channel_2.Status/Overrange <-> AI Standard Channel 2/Status/Overrange
//     PlcTask Inputs/GVL_iXlinker.EtherCAT_Master_EJxxxx.Beckhoff_EJ3xxx.A_0003_EJ3004_0000_0021.AI_Standard_Channel_3.Status/Overrange <-> AI Standard Channel 3/Status/Overrange
//     PlcTask Inputs/GVL_iXlinker.EtherCAT_Master_EJxxxx.Beckhoff_EJ3xxx.A_0003_EJ3004_0000_0021.AI_Standard_Channel_4.Status/Overrange <-> AI Standard Channel 4/Status/Overrange
//     PlcTask Inputs/GVL_iXlinker.EtherCAT_Master_EJxxxx.Beckhoff_EJ3xxx.A_0003_EJ3004_0000_0021.AI_Standard_Channel_1.Status/Limit_1 <-> AI Standard Channel 1/Status/Limit 1
//     PlcTask Inputs/GVL_iXlinker.EtherCAT_Master_EJxxxx.Beckhoff_EJ3xxx.A_0003_EJ3004_0000_0021.AI_Standard_Channel_1.Status/Limit_2 <-> AI Standard Channel 1/Status/Limit 2
//     PlcTask Inputs/GVL_iXlinker.EtherCAT_Master_EJxxxx.Beckhoff_EJ3xxx.A_0003_EJ3004_0000_0021.AI_Standard_Channel_2.Status/Limit_1 <-> AI Standard Channel 2/Status/Limit 1
//     PlcTask Inputs/GVL_iXlinker.EtherCAT_Master_EJxxxx.Beckhoff_EJ3xxx.A_0003_EJ3004_0000_0021.AI_Standard_Channel_2.Status/Limit_2 <-> AI Standard Channel 2/Status/Limit 2
//     PlcTask Inputs/GVL_iXlinker.EtherCAT_Master_EJxxxx.Beckhoff_EJ3xxx.A_0003_EJ3004_0000_0021.AI_Standard_Channel_3.Status/Limit_1 <-> AI Standard Channel 3/Status/Limit 1
//     PlcTask Inputs/GVL_iXlinker.EtherCAT_Master_EJxxxx.Beckhoff_EJ3xxx.A_0003_EJ3004_0000_0021.AI_Standard_Channel_3.Status/Limit_2 <-> AI Standard Channel 3/Status/Limit 2
//     PlcTask Inputs/GVL_iXlinker.EtherCAT_Master_EJxxxx.Beckhoff_EJ3xxx.A_0003_EJ3004_0000_0021.AI_Standard_Channel_4.Status/Limit_1 <-> AI Standard Channel 4/Status/Limit 1
//     PlcTask Inputs/GVL_iXlinker.EtherCAT_Master_EJxxxx.Beckhoff_EJ3xxx.A_0003_EJ3004_0000_0021.AI_Standard_Channel_4.Status/Limit_2 <-> AI Standard Channel 4/Status/Limit 2
//     PlcTask Inputs/GVL_iXlinker.EtherCAT_Master_EJxxxx.Beckhoff_EJ3xxx.A_0003_EJ3004_0000_0021.AI_Standard_Channel_1.Status/Error <-> AI Standard Channel 1/Status/Error
//     PlcTask Inputs/GVL_iXlinker.EtherCAT_Master_EJxxxx.Beckhoff_EJ3xxx.A_0003_EJ3004_0000_0021.AI_Standard_Channel_2.Status/Error <-> AI Standard Channel 2/Status/Error
//     PlcTask Inputs/GVL_iXlinker.EtherCAT_Master_EJxxxx.Beckhoff_EJ3xxx.A_0003_EJ3004_0000_0021.AI_Standard_Channel_3.Status/Error <-> AI Standard Channel 3/Status/Error
//     PlcTask Inputs/GVL_iXlinker.EtherCAT_Master_EJxxxx.Beckhoff_EJ3xxx.A_0003_EJ3004_0000_0021.AI_Standard_Channel_4.Status/Error <-> AI Standard Channel 4/Status/Error
//     PlcTask Inputs/GVL_iXlinker.EtherCAT_Master_EJxxxx.Beckhoff_EJ3xxx.A_0003_EJ3004_0000_0021.AI_Standard_Channel_1.Status/TxPDO_State <-> AI Standard Channel 1/Status/TxPDO State
//     PlcTask Inputs/GVL_iXlinker.EtherCAT_Master_EJxxxx.Beckhoff_EJ3xxx.A_0003_EJ3004_0000_0021.AI_Standard_Channel_2.Status/TxPDO_State <-> AI Standard Channel 2/Status/TxPDO State
//     PlcTask Inputs/GVL_iXlinker.EtherCAT_Master_EJxxxx.Beckhoff_EJ3xxx.A_0003_EJ3004_0000_0021.AI_Standard_Channel_3.Status/TxPDO_State <-> AI Standard Channel 3/Status/TxPDO State
//     PlcTask Inputs/GVL_iXlinker.EtherCAT_Master_EJxxxx.Beckhoff_EJ3xxx.A_0003_EJ3004_0000_0021.AI_Standard_Channel_4.Status/TxPDO_State <-> AI Standard Channel 4/Status/TxPDO State
//     PlcTask Inputs/GVL_iXlinker.EtherCAT_Master_EJxxxx.Beckhoff_EJ3xxx.A_0003_EJ3004_0000_0021.AI_Standard_Channel_1.Status/TxPDO_Toggle <-> AI Standard Channel 1/Status/TxPDO Toggle
//     PlcTask Inputs/GVL_iXlinker.EtherCAT_Master_EJxxxx.Beckhoff_EJ3xxx.A_0003_EJ3004_0000_0021.AI_Standard_Channel_2.Status/TxPDO_Toggle <-> AI Standard Channel 2/Status/TxPDO Toggle
//     PlcTask Inputs/GVL_iXlinker.EtherCAT_Master_EJxxxx.Beckhoff_EJ3xxx.A_0003_EJ3004_0000_0021.AI_Standard_Channel_3.Status/TxPDO_Toggle <-> AI Standard Channel 3/Status/TxPDO Toggle
//     PlcTask Inputs/GVL_iXlinker.EtherCAT_Master_EJxxxx.Beckhoff_EJ3xxx.A_0003_EJ3004_0000_0021.AI_Standard_Channel_4.Status/TxPDO_Toggle <-> AI Standard Channel 4/Status/TxPDO Toggle
//     PlcTask Inputs/GVL_iXlinker.EtherCAT_Master_EJxxxx.Beckhoff_EJ3xxx.A_0003_EJ3004_0000_0021.AI_Standard_Channel_1.Value <-> AI Standard Channel 1/Value
//     PlcTask Inputs/GVL_iXlinker.EtherCAT_Master_EJxxxx.Beckhoff_EJ3xxx.A_0003_EJ3004_0000_0021.AI_Standard_Channel_2.Value <-> AI Standard Channel 2/Value
//     PlcTask Inputs/GVL_iXlinker.EtherCAT_Master_EJxxxx.Beckhoff_EJ3xxx.A_0003_EJ3004_0000_0021.AI_Standard_Channel_3.Value <-> AI Standard Channel 3/Value
//     PlcTask Inputs/GVL_iXlinker.EtherCAT_Master_EJxxxx.Beckhoff_EJ3xxx.A_0003_EJ3004_0000_0021.AI_Standard_Channel_4.Value <-> AI Standard Channel 4/Value
//     PlcTask Inputs/GVL_iXlinker.EtherCAT_Master_EJxxxx.Beckhoff_EJ3xxx.A_0003_EJ3004_0000_0021.WcState.WcState <-> WcState/WcState
//     PlcTask Inputs/GVL_iXlinker.EtherCAT_Master_EJxxxx.Beckhoff_EJ3xxx.A_0003_EJ3004_0000_0021.WcState.InputToggle <-> WcState/InputToggle
//     PlcTask Inputs/GVL_iXlinker.EtherCAT_Master_EJxxxx.Beckhoff_EJ3xxx.A_0003_EJ3004_0000_0021.InfoData.AdsAddr <-> InfoData/AdsAddr
//     PlcTask Inputs/GVL_iXlinker.EtherCAT_Master_EJxxxx.Beckhoff_EJ3xxx.A_0003_EJ3004_0000_0021.InfoData.State <-> InfoData/State
//   PLC/PLC Instance <-> EtherCAT Master EJxxxx/Beckhoff EJ3xxx/A_0004(EJ3048-0000-0020)
//     PlcTask Inputs/GVL_iXlinker.EtherCAT_Master_EJxxxx.Beckhoff_EJ3xxx.A_0004_EJ3048_0000_0020.AI_Standard_Channel_1.Status/Underrange <-> AI Standard Channel 1/Status/Underrange
//     PlcTask Inputs/GVL_iXlinker.EtherCAT_Master_EJxxxx.Beckhoff_EJ3xxx.A_0004_EJ3048_0000_0020.AI_Standard_Channel_2.Status/Underrange <-> AI Standard Channel 2/Status/Underrange
//     PlcTask Inputs/GVL_iXlinker.EtherCAT_Master_EJxxxx.Beckhoff_EJ3xxx.A_0004_EJ3048_0000_0020.AI_Standard_Channel_3.Status/Underrange <-> AI Standard Channel 3/Status/Underrange
//     PlcTask Inputs/GVL_iXlinker.EtherCAT_Master_EJxxxx.Beckhoff_EJ3xxx.A_0004_EJ3048_0000_0020.AI_Standard_Channel_4.Status/Underrange <-> AI Standard Channel 4/Status/Underrange
//     PlcTask Inputs/GVL_iXlinker.EtherCAT_Master_EJxxxx.Beckhoff_EJ3xxx.A_0004_EJ3048_0000_0020.AI_Standard_Channel_5.Status/Underrange <-> AI Standard Channel 5/Status/Underrange
//     PlcTask Inputs/GVL_iXlinker.EtherCAT_Master_EJxxxx.Beckhoff_EJ3xxx.A_0004_EJ3048_0000_0020.AI_Standard_Channel_6.Status/Underrange <-> AI Standard Channel 6/Status/Underrange
//     PlcTask Inputs/GVL_iXlinker.EtherCAT_Master_EJxxxx.Beckhoff_EJ3xxx.A_0004_EJ3048_0000_0020.AI_Standard_Channel_7.Status/Underrange <-> AI Standard Channel 7/Status/Underrange
//     PlcTask Inputs/GVL_iXlinker.EtherCAT_Master_EJxxxx.Beckhoff_EJ3xxx.A_0004_EJ3048_0000_0020.AI_Standard_Channel_8.Status/Underrange <-> AI Standard Channel 8/Status/Underrange
//     PlcTask Inputs/GVL_iXlinker.EtherCAT_Master_EJxxxx.Beckhoff_EJ3xxx.A_0004_EJ3048_0000_0020.AI_Standard_Channel_1.Status/Overrange <-> AI Standard Channel 1/Status/Overrange
//     PlcTask Inputs/GVL_iXlinker.EtherCAT_Master_EJxxxx.Beckhoff_EJ3xxx.A_0004_EJ3048_0000_0020.AI_Standard_Channel_2.Status/Overrange <-> AI Standard Channel 2/Status/Overrange
//     PlcTask Inputs/GVL_iXlinker.EtherCAT_Master_EJxxxx.Beckhoff_EJ3xxx.A_0004_EJ3048_0000_0020.AI_Standard_Channel_3.Status/Overrange <-> AI Standard Channel 3/Status/Overrange
//     PlcTask Inputs/GVL_iXlinker.EtherCAT_Master_EJxxxx.Beckhoff_EJ3xxx.A_0004_EJ3048_0000_0020.AI_Standard_Channel_4.Status/Overrange <-> AI Standard Channel 4/Status/Overrange
//     PlcTask Inputs/GVL_iXlinker.EtherCAT_Master_EJxxxx.Beckhoff_EJ3xxx.A_0004_EJ3048_0000_0020.AI_Standard_Channel_5.Status/Overrange <-> AI Standard Channel 5/Status/Overrange
//     PlcTask Inputs/GVL_iXlinker.EtherCAT_Master_EJxxxx.Beckhoff_EJ3xxx.A_0004_EJ3048_0000_0020.AI_Standard_Channel_6.Status/Overrange <-> AI Standard Channel 6/Status/Overrange
//     PlcTask Inputs/GVL_iXlinker.EtherCAT_Master_EJxxxx.Beckhoff_EJ3xxx.A_0004_EJ3048_0000_0020.AI_Standard_Channel_7.Status/Overrange <-> AI Standard Channel 7/Status/Overrange
//     PlcTask Inputs/GVL_iXlinker.EtherCAT_Master_EJxxxx.Beckhoff_EJ3xxx.A_0004_EJ3048_0000_0020.AI_Standard_Channel_8.Status/Overrange <-> AI Standard Channel 8/Status/Overrange
//     PlcTask Inputs/GVL_iXlinker.EtherCAT_Master_EJxxxx.Beckhoff_EJ3xxx.A_0004_EJ3048_0000_0020.AI_Standard_Channel_1.Status/Limit_1 <-> AI Standard Channel 1/Status/Limit 1
//     PlcTask Inputs/GVL_iXlinker.EtherCAT_Master_EJxxxx.Beckhoff_EJ3xxx.A_0004_EJ3048_0000_0020.AI_Standard_Channel_1.Status/Limit_2 <-> AI Standard Channel 1/Status/Limit 2
//     PlcTask Inputs/GVL_iXlinker.EtherCAT_Master_EJxxxx.Beckhoff_EJ3xxx.A_0004_EJ3048_0000_0020.AI_Standard_Channel_2.Status/Limit_1 <-> AI Standard Channel 2/Status/Limit 1
//     PlcTask Inputs/GVL_iXlinker.EtherCAT_Master_EJxxxx.Beckhoff_EJ3xxx.A_0004_EJ3048_0000_0020.AI_Standard_Channel_2.Status/Limit_2 <-> AI Standard Channel 2/Status/Limit 2
//     PlcTask Inputs/GVL_iXlinker.EtherCAT_Master_EJxxxx.Beckhoff_EJ3xxx.A_0004_EJ3048_0000_0020.AI_Standard_Channel_3.Status/Limit_1 <-> AI Standard Channel 3/Status/Limit 1
//     PlcTask Inputs/GVL_iXlinker.EtherCAT_Master_EJxxxx.Beckhoff_EJ3xxx.A_0004_EJ3048_0000_0020.AI_Standard_Channel_3.Status/Limit_2 <-> AI Standard Channel 3/Status/Limit 2
//     PlcTask Inputs/GVL_iXlinker.EtherCAT_Master_EJxxxx.Beckhoff_EJ3xxx.A_0004_EJ3048_0000_0020.AI_Standard_Channel_4.Status/Limit_1 <-> AI Standard Channel 4/Status/Limit 1
//     PlcTask Inputs/GVL_iXlinker.EtherCAT_Master_EJxxxx.Beckhoff_EJ3xxx.A_0004_EJ3048_0000_0020.AI_Standard_Channel_4.Status/Limit_2 <-> AI Standard Channel 4/Status/Limit 2
//     PlcTask Inputs/GVL_iXlinker.EtherCAT_Master_EJxxxx.Beckhoff_EJ3xxx.A_0004_EJ3048_0000_0020.AI_Standard_Channel_5.Status/Limit_1 <-> AI Standard Channel 5/Status/Limit 1
//     PlcTask Inputs/GVL_iXlinker.EtherCAT_Master_EJxxxx.Beckhoff_EJ3xxx.A_0004_EJ3048_0000_0020.AI_Standard_Channel_5.Status/Limit_2 <-> AI Standard Channel 5/Status/Limit 2
//     PlcTask Inputs/GVL_iXlinker.EtherCAT_Master_EJxxxx.Beckhoff_EJ3xxx.A_0004_EJ3048_0000_0020.AI_Standard_Channel_6.Status/Limit_1 <-> AI Standard Channel 6/Status/Limit 1
//     PlcTask Inputs/GVL_iXlinker.EtherCAT_Master_EJxxxx.Beckhoff_EJ3xxx.A_0004_EJ3048_0000_0020.AI_Standard_Channel_6.Status/Limit_2 <-> AI Standard Channel 6/Status/Limit 2
//     PlcTask Inputs/GVL_iXlinker.EtherCAT_Master_EJxxxx.Beckhoff_EJ3xxx.A_0004_EJ3048_0000_0020.AI_Standard_Channel_7.Status/Limit_1 <-> AI Standard Channel 7/Status/Limit 1
//     PlcTask Inputs/GVL_iXlinker.EtherCAT_Master_EJxxxx.Beckhoff_EJ3xxx.A_0004_EJ3048_0000_0020.AI_Standard_Channel_7.Status/Limit_2 <-> AI Standard Channel 7/Status/Limit 2
//     PlcTask Inputs/GVL_iXlinker.EtherCAT_Master_EJxxxx.Beckhoff_EJ3xxx.A_0004_EJ3048_0000_0020.AI_Standard_Channel_8.Status/Limit_1 <-> AI Standard Channel 8/Status/Limit 1
//     PlcTask Inputs/GVL_iXlinker.EtherCAT_Master_EJxxxx.Beckhoff_EJ3xxx.A_0004_EJ3048_0000_0020.AI_Standard_Channel_8.Status/Limit_2 <-> AI Standard Channel 8/Status/Limit 2
//     PlcTask Inputs/GVL_iXlinker.EtherCAT_Master_EJxxxx.Beckhoff_EJ3xxx.A_0004_EJ3048_0000_0020.AI_Standard_Channel_1.Status/Error <-> AI Standard Channel 1/Status/Error
//     PlcTask Inputs/GVL_iXlinker.EtherCAT_Master_EJxxxx.Beckhoff_EJ3xxx.A_0004_EJ3048_0000_0020.AI_Standard_Channel_2.Status/Error <-> AI Standard Channel 2/Status/Error
//     PlcTask Inputs/GVL_iXlinker.EtherCAT_Master_EJxxxx.Beckhoff_EJ3xxx.A_0004_EJ3048_0000_0020.AI_Standard_Channel_3.Status/Error <-> AI Standard Channel 3/Status/Error
//     PlcTask Inputs/GVL_iXlinker.EtherCAT_Master_EJxxxx.Beckhoff_EJ3xxx.A_0004_EJ3048_0000_0020.AI_Standard_Channel_4.Status/Error <-> AI Standard Channel 4/Status/Error
//     PlcTask Inputs/GVL_iXlinker.EtherCAT_Master_EJxxxx.Beckhoff_EJ3xxx.A_0004_EJ3048_0000_0020.AI_Standard_Channel_5.Status/Error <-> AI Standard Channel 5/Status/Error
//     PlcTask Inputs/GVL_iXlinker.EtherCAT_Master_EJxxxx.Beckhoff_EJ3xxx.A_0004_EJ3048_0000_0020.AI_Standard_Channel_6.Status/Error <-> AI Standard Channel 6/Status/Error
//     PlcTask Inputs/GVL_iXlinker.EtherCAT_Master_EJxxxx.Beckhoff_EJ3xxx.A_0004_EJ3048_0000_0020.AI_Standard_Channel_7.Status/Error <-> AI Standard Channel 7/Status/Error
//     PlcTask Inputs/GVL_iXlinker.EtherCAT_Master_EJxxxx.Beckhoff_EJ3xxx.A_0004_EJ3048_0000_0020.AI_Standard_Channel_8.Status/Error <-> AI Standard Channel 8/Status/Error
//     PlcTask Inputs/GVL_iXlinker.EtherCAT_Master_EJxxxx.Beckhoff_EJ3xxx.A_0004_EJ3048_0000_0020.AI_Standard_Channel_1.Status/TxPDO_State <-> AI Standard Channel 1/Status/TxPDO State
//     PlcTask Inputs/GVL_iXlinker.EtherCAT_Master_EJxxxx.Beckhoff_EJ3xxx.A_0004_EJ3048_0000_0020.AI_Standard_Channel_2.Status/TxPDO_State <-> AI Standard Channel 2/Status/TxPDO State
//     PlcTask Inputs/GVL_iXlinker.EtherCAT_Master_EJxxxx.Beckhoff_EJ3xxx.A_0004_EJ3048_0000_0020.AI_Standard_Channel_3.Status/TxPDO_State <-> AI Standard Channel 3/Status/TxPDO State
//     PlcTask Inputs/GVL_iXlinker.EtherCAT_Master_EJxxxx.Beckhoff_EJ3xxx.A_0004_EJ3048_0000_0020.AI_Standard_Channel_4.Status/TxPDO_State <-> AI Standard Channel 4/Status/TxPDO State
//     PlcTask Inputs/GVL_iXlinker.EtherCAT_Master_EJxxxx.Beckhoff_EJ3xxx.A_0004_EJ3048_0000_0020.AI_Standard_Channel_5.Status/TxPDO_State <-> AI Standard Channel 5/Status/TxPDO State
//     PlcTask Inputs/GVL_iXlinker.EtherCAT_Master_EJxxxx.Beckhoff_EJ3xxx.A_0004_EJ3048_0000_0020.AI_Standard_Channel_6.Status/TxPDO_State <-> AI Standard Channel 6/Status/TxPDO State
//     PlcTask Inputs/GVL_iXlinker.EtherCAT_Master_EJxxxx.Beckhoff_EJ3xxx.A_0004_EJ3048_0000_0020.AI_Standard_Channel_7.Status/TxPDO_State <-> AI Standard Channel 7/Status/TxPDO State
//     PlcTask Inputs/GVL_iXlinker.EtherCAT_Master_EJxxxx.Beckhoff_EJ3xxx.A_0004_EJ3048_0000_0020.AI_Standard_Channel_8.Status/TxPDO_State <-> AI Standard Channel 8/Status/TxPDO State
//     PlcTask Inputs/GVL_iXlinker.EtherCAT_Master_EJxxxx.Beckhoff_EJ3xxx.A_0004_EJ3048_0000_0020.AI_Standard_Channel_1.Status/TxPDO_Toggle <-> AI Standard Channel 1/Status/TxPDO Toggle
//     PlcTask Inputs/GVL_iXlinker.EtherCAT_Master_EJxxxx.Beckhoff_EJ3xxx.A_0004_EJ3048_0000_0020.AI_Standard_Channel_2.Status/TxPDO_Toggle <-> AI Standard Channel 2/Status/TxPDO Toggle
//     PlcTask Inputs/GVL_iXlinker.EtherCAT_Master_EJxxxx.Beckhoff_EJ3xxx.A_0004_EJ3048_0000_0020.AI_Standard_Channel_3.Status/TxPDO_Toggle <-> AI Standard Channel 3/Status/TxPDO Toggle
//     PlcTask Inputs/GVL_iXlinker.EtherCAT_Master_EJxxxx.Beckhoff_EJ3xxx.A_0004_EJ3048_0000_0020.AI_Standard_Channel_4.Status/TxPDO_Toggle <-> AI Standard Channel 4/Status/TxPDO Toggle
//     PlcTask Inputs/GVL_iXlinker.EtherCAT_Master_EJxxxx.Beckhoff_EJ3xxx.A_0004_EJ3048_0000_0020.AI_Standard_Channel_5.Status/TxPDO_Toggle <-> AI Standard Channel 5/Status/TxPDO Toggle
//     PlcTask Inputs/GVL_iXlinker.EtherCAT_Master_EJxxxx.Beckhoff_EJ3xxx.A_0004_EJ3048_0000_0020.AI_Standard_Channel_6.Status/TxPDO_Toggle <-> AI Standard Channel 6/Status/TxPDO Toggle
//     PlcTask Inputs/GVL_iXlinker.EtherCAT_Master_EJxxxx.Beckhoff_EJ3xxx.A_0004_EJ3048_0000_0020.AI_Standard_Channel_7.Status/TxPDO_Toggle <-> AI Standard Channel 7/Status/TxPDO Toggle
//     PlcTask Inputs/GVL_iXlinker.EtherCAT_Master_EJxxxx.Beckhoff_EJ3xxx.A_0004_EJ3048_0000_0020.AI_Standard_Channel_8.Status/TxPDO_Toggle <-> AI Standard Channel 8/Status/TxPDO Toggle
//     PlcTask Inputs/GVL_iXlinker.EtherCAT_Master_EJxxxx.Beckhoff_EJ3xxx.A_0004_EJ3048_0000_0020.AI_Standard_Channel_1.Value <-> AI Standard Channel 1/Value
//     PlcTask Inputs/GVL_iXlinker.EtherCAT_Master_EJxxxx.Beckhoff_EJ3xxx.A_0004_EJ3048_0000_0020.AI_Standard_Channel_2.Value <-> AI Standard Channel 2/Value
//     PlcTask Inputs/GVL_iXlinker.EtherCAT_Master_EJxxxx.Beckhoff_EJ3xxx.A_0004_EJ3048_0000_0020.AI_Standard_Channel_3.Value <-> AI Standard Channel 3/Value
//     PlcTask Inputs/GVL_iXlinker.EtherCAT_Master_EJxxxx.Beckhoff_EJ3xxx.A_0004_EJ3048_0000_0020.AI_Standard_Channel_4.Value <-> AI Standard Channel 4/Value
//     PlcTask Inputs/GVL_iXlinker.EtherCAT_Master_EJxxxx.Beckhoff_EJ3xxx.A_0004_EJ3048_0000_0020.AI_Standard_Channel_5.Value <-> AI Standard Channel 5/Value
//     PlcTask Inputs/GVL_iXlinker.EtherCAT_Master_EJxxxx.Beckhoff_EJ3xxx.A_0004_EJ3048_0000_0020.AI_Standard_Channel_6.Value <-> AI Standard Channel 6/Value
//     PlcTask Inputs/GVL_iXlinker.EtherCAT_Master_EJxxxx.Beckhoff_EJ3xxx.A_0004_EJ3048_0000_0020.AI_Standard_Channel_7.Value <-> AI Standard Channel 7/Value
//     PlcTask Inputs/GVL_iXlinker.EtherCAT_Master_EJxxxx.Beckhoff_EJ3xxx.A_0004_EJ3048_0000_0020.AI_Standard_Channel_8.Value <-> AI Standard Channel 8/Value
//     PlcTask Inputs/GVL_iXlinker.EtherCAT_Master_EJxxxx.Beckhoff_EJ3xxx.A_0004_EJ3048_0000_0020.WcState.WcState <-> WcState/WcState
//     PlcTask Inputs/GVL_iXlinker.EtherCAT_Master_EJxxxx.Beckhoff_EJ3xxx.A_0004_EJ3048_0000_0020.WcState.InputToggle <-> WcState/InputToggle
//     PlcTask Inputs/GVL_iXlinker.EtherCAT_Master_EJxxxx.Beckhoff_EJ3xxx.A_0004_EJ3048_0000_0020.InfoData.AdsAddr <-> InfoData/AdsAddr
//     PlcTask Inputs/GVL_iXlinker.EtherCAT_Master_EJxxxx.Beckhoff_EJ3xxx.A_0004_EJ3048_0000_0020.InfoData.State <-> InfoData/State
//   PLC/PLC Instance <-> EtherCAT Master EJxxxx/Beckhoff EJ3xxx/A_0005(EJ3058-0000-0020)
//     PlcTask Inputs/GVL_iXlinker.EtherCAT_Master_EJxxxx.Beckhoff_EJ3xxx.A_0005_EJ3058_0000_0020.AI_Standard_Channel_1.Status/Underrange <-> AI Standard Channel 1/Status/Underrange
//     PlcTask Inputs/GVL_iXlinker.EtherCAT_Master_EJxxxx.Beckhoff_EJ3xxx.A_0005_EJ3058_0000_0020.AI_Standard_Channel_2.Status/Underrange <-> AI Standard Channel 2/Status/Underrange
//     PlcTask Inputs/GVL_iXlinker.EtherCAT_Master_EJxxxx.Beckhoff_EJ3xxx.A_0005_EJ3058_0000_0020.AI_Standard_Channel_3.Status/Underrange <-> AI Standard Channel 3/Status/Underrange
//     PlcTask Inputs/GVL_iXlinker.EtherCAT_Master_EJxxxx.Beckhoff_EJ3xxx.A_0005_EJ3058_0000_0020.AI_Standard_Channel_4.Status/Underrange <-> AI Standard Channel 4/Status/Underrange
//     PlcTask Inputs/GVL_iXlinker.EtherCAT_Master_EJxxxx.Beckhoff_EJ3xxx.A_0005_EJ3058_0000_0020.AI_Standard_Channel_5.Status/Underrange <-> AI Standard Channel 5/Status/Underrange
//     PlcTask Inputs/GVL_iXlinker.EtherCAT_Master_EJxxxx.Beckhoff_EJ3xxx.A_0005_EJ3058_0000_0020.AI_Standard_Channel_6.Status/Underrange <-> AI Standard Channel 6/Status/Underrange
//     PlcTask Inputs/GVL_iXlinker.EtherCAT_Master_EJxxxx.Beckhoff_EJ3xxx.A_0005_EJ3058_0000_0020.AI_Standard_Channel_7.Status/Underrange <-> AI Standard Channel 7/Status/Underrange
//     PlcTask Inputs/GVL_iXlinker.EtherCAT_Master_EJxxxx.Beckhoff_EJ3xxx.A_0005_EJ3058_0000_0020.AI_Standard_Channel_8.Status/Underrange <-> AI Standard Channel 8/Status/Underrange
//     PlcTask Inputs/GVL_iXlinker.EtherCAT_Master_EJxxxx.Beckhoff_EJ3xxx.A_0005_EJ3058_0000_0020.AI_Standard_Channel_1.Status/Overrange <-> AI Standard Channel 1/Status/Overrange
//     PlcTask Inputs/GVL_iXlinker.EtherCAT_Master_EJxxxx.Beckhoff_EJ3xxx.A_0005_EJ3058_0000_0020.AI_Standard_Channel_2.Status/Overrange <-> AI Standard Channel 2/Status/Overrange
//     PlcTask Inputs/GVL_iXlinker.EtherCAT_Master_EJxxxx.Beckhoff_EJ3xxx.A_0005_EJ3058_0000_0020.AI_Standard_Channel_3.Status/Overrange <-> AI Standard Channel 3/Status/Overrange
//     PlcTask Inputs/GVL_iXlinker.EtherCAT_Master_EJxxxx.Beckhoff_EJ3xxx.A_0005_EJ3058_0000_0020.AI_Standard_Channel_4.Status/Overrange <-> AI Standard Channel 4/Status/Overrange
//     PlcTask Inputs/GVL_iXlinker.EtherCAT_Master_EJxxxx.Beckhoff_EJ3xxx.A_0005_EJ3058_0000_0020.AI_Standard_Channel_5.Status/Overrange <-> AI Standard Channel 5/Status/Overrange
//     PlcTask Inputs/GVL_iXlinker.EtherCAT_Master_EJxxxx.Beckhoff_EJ3xxx.A_0005_EJ3058_0000_0020.AI_Standard_Channel_6.Status/Overrange <-> AI Standard Channel 6/Status/Overrange
//     PlcTask Inputs/GVL_iXlinker.EtherCAT_Master_EJxxxx.Beckhoff_EJ3xxx.A_0005_EJ3058_0000_0020.AI_Standard_Channel_7.Status/Overrange <-> AI Standard Channel 7/Status/Overrange
//     PlcTask Inputs/GVL_iXlinker.EtherCAT_Master_EJxxxx.Beckhoff_EJ3xxx.A_0005_EJ3058_0000_0020.AI_Standard_Channel_8.Status/Overrange <-> AI Standard Channel 8/Status/Overrange
//     PlcTask Inputs/GVL_iXlinker.EtherCAT_Master_EJxxxx.Beckhoff_EJ3xxx.A_0005_EJ3058_0000_0020.AI_Standard_Channel_1.Status/Limit_1 <-> AI Standard Channel 1/Status/Limit 1
//     PlcTask Inputs/GVL_iXlinker.EtherCAT_Master_EJxxxx.Beckhoff_EJ3xxx.A_0005_EJ3058_0000_0020.AI_Standard_Channel_1.Status/Limit_2 <-> AI Standard Channel 1/Status/Limit 2
//     PlcTask Inputs/GVL_iXlinker.EtherCAT_Master_EJxxxx.Beckhoff_EJ3xxx.A_0005_EJ3058_0000_0020.AI_Standard_Channel_2.Status/Limit_1 <-> AI Standard Channel 2/Status/Limit 1
//     PlcTask Inputs/GVL_iXlinker.EtherCAT_Master_EJxxxx.Beckhoff_EJ3xxx.A_0005_EJ3058_0000_0020.AI_Standard_Channel_2.Status/Limit_2 <-> AI Standard Channel 2/Status/Limit 2
//     PlcTask Inputs/GVL_iXlinker.EtherCAT_Master_EJxxxx.Beckhoff_EJ3xxx.A_0005_EJ3058_0000_0020.AI_Standard_Channel_3.Status/Limit_1 <-> AI Standard Channel 3/Status/Limit 1
